	nu_On:			CustomPhase (table:=ADR(phasesTable)):=			(phaseNumber:=24);
	flag1:BOOL;
	Start_AO_From:			CustomPhase (table:=ADR(phasesTable)):=			(phaseNumber:=25);
END_VAR

SUPER^();

//////////////Старт смазки кранов 1 и 2///////////////////////////
IF	algoritms.F3.Smazka_1_2 OR (im.kran1.onStatus = statusDualInput.STATUS_ON) OR (im.kran1.onStatus = statusDualInput.STATUS_TRANSITIONAL)
	OR (im.kran2.onStatus = statusDualInput.STATUS_ON) OR (im.kran2.onStatus = statusDualInput.STATUS_TRANSITIONAL)  THEN
	IF	(algoritms.F3.Smazka_1_2 OR (im.kran1.onStatus = statusDualInput.STATUS_ON) OR (im.kran1.onStatus = statusDualInput.STATUS_TRANSITIONAL)) AND (NOT klapan1.start) AND (NOT kran1Close.top) THEN
		klapan1.run ();
	END_IF
	IF	(algoritms.F3.Smazka_1_2 OR (im.kran2.onStatus = statusDualInput.STATUS_ON) OR (im.kran2.onStatus = statusDualInput.STATUS_TRANSITIONAL)) AND (NOT klapan2.start) AND (NOT kran2Close.top) THEN
		klapan2.run ();
	END_IF
	algoritms.F3.Smazka_1_2:=FALSE;
END_IF

//////////////Переставляем краны///////////////////////////
IF	NOT kran6Open.start THEN
	ystavki.Block_kr6_alg.setValue (1);
	IF	im.kran6._cmdreset.IN = FALSE THEN
		ystavki.Block_kr6_alg.setValue (0);
		kran6Open.run(); //открываем карн 6
	END_IF
END_IF

IF	NOT kran4Close.start THEN
	ystavki.Block_kr4_alg.setValue (1);
	IF	im.kran4._cmdreset.IN = FALSE THEN
		ystavki.Block_kr4_alg.setValue (0);
		kran4Close.run(); //закрываем кран 4
	END_IF
END_IF

IF	NOT kran3bOpen.start THEN
	ystavki.Block_kr3b_alg.setValue (1);
	IF	im.kran3b._cmdreset.IN = FALSE THEN
		ystavki.Block_kr3b_alg.setValue (0);
		kran3bOpen.run (); //Открываем кран 3бис
	END_IF
END_IF
protections.p_mvOff.reset ();
protections.p_OFFAvarSwitch.reset();
protections.p_RegVozbOff.reset ();
protections.p_kran1.reset ();
protections.p_kran2.reset ();
mvOff.run(); //отключаем МВ

IF	NOT kran1Close.start THEN
	ystavki.Block_kr1_alg.setValue (1);
	IF	im.kran1._cmdreset.IN = FALSE THEN
		ystavki.Block_kr1_alg.setValue (0);
		kran1Close.run(); //закрываем кран 1
	END_IF
END_IF

IF	NOT	kran2Close.start THEN
	ystavki.Block_kr2_alg.setValue (1);
	IF	im.kran2._cmdreset.IN = FALSE THEN
		ystavki.Block_kr2_alg.setValue (0);
		kran2Close.run(); //закрываем кран 2 
	END_IF
END_IF

IF	NOT	kran3Close.start THEN
	ystavki.Block_kr3_alg.setValue (1);
	IF	im.kran3._cmdreset.IN = FALSE THEN
		ystavki.Block_kr3_alg.setValue (0);
		kran3Close.run(); //закрываем кран 3
	END_IF
END_IF

IF	kran6Open.top THEN
	algoritms.S_Vibr.CanRun:=FALSE;
	algoritms.S_Vibr.reset ();
END_IF
///////////////выдаем смазку кранов 1 и 2//////////////////////////
IF	klapan1.start AND kran1Close.top THEN
	im.Kr1_Smazka.impulse();//выдача команды на клапан
	klapan1.top:=TRUE;
END_IF;
IF	klapan2.start AND kran2Close.top THEN
	im.Kr2_Smazka.impulse();//выдача команды на клапан
	klapan2.top:=TRUE;
END_IF;
///////////////открываем кран 5//////////////////////////
IF 	kran1Close.top AND kran2Close.top AND kran3Close.top AND kran4Close.top AND NOT kran5Open.top THEN //если кран 1 и 2 закрыты открываем кран 5
	IF	NOT	kran5Open.start THEN
		ystavki.Block_kr5_alg.setValue (1);
		IF	im.kran5._cmdreset.IN = FALSE THEN
			ystavki.Block_kr5_alg.setValue (0);
			kran5Open.run();
		END_IF
	END_IF

	//protections.p_DGazaNaVhodeNagnetatelja.reset ();
	protections.p_DGazaNaVyhodeNagnetatelja.reset ();
END_IF 
/////////////////////////////////////////
IF	mvOff.top AND NOT flag1 THEN //если МВ отключился 
	algoritms.AutoPNS_Start.canrun :=FALSE;
	algoritms.AutoPNS_Start.reset ();
	algoritms.autoPns.canrun :=FALSE;
	autoPnsOff.run ();
	pnsOn.run ();
	nu_On.run();
	CASE 	im.nu.mainNasos.Value OF
	0:		im.nu.nu1.on ();
	1:		im.nu.nu2.on ();
	END_CASE
	algoritms.autoNu_2.canrun:=FALSE;
	algoritms.autoNu_2.reset ();
	algoritms.autoNu_1.canrun:=TRUE;
	algoritms.autoNu_1.run ();
	flag1:=TRUE;
END_IF
IF	((im.nu.nu1.onStatus =statusDualInput.STATUS_On) OR (im.nu.nu2.onStatus =statusDualInput.STATUS_On)) AND nu_On.start AND NOT nu_On.top THEN
	nu_On.top:=TRUE;
END_IF
/////////////////////////////////////////
IF 	kran5Open.top THEN //если отключены МВ и 5 кран
	Pg_VhodLessThen300.run();  //проверяем условие, что давление в нагнетателе меньше 100
	Pg_VyhodLessThen300.run(); 
	
END_IF 
/////////////////////////////////////////
IF Pg_VhodLessThen300.start AND (NOT Pg_VhodLessThen300.top) THEN
	IF 	(ai.DGazaNaVhodeNagnetatelja.interval>=statusAi.NORMAL) AND (ai.DGazaNaVhodeNagnetatelja.value < 0.3 )THEN
		Pg_VhodLessThen300.top:=TRUE; //давление в полости нагнетателя меньше 100 кПа
	END_IF
END_IF
/////////////////////////////////////////
IF Pg_VyhodLessThen300.start AND (NOT Pg_VyhodLessThen300.top) THEN
	IF 	(ai.DGazaNaVyhodeNagnetatelja.interval>=statusAi.NORMAL) AND (ai.DGazaNaVyhodeNagnetatelja.value < 0.3) THEN
		Pg_VyhodLessThen300.top:=TRUE; //давление в полости нагнетателя меньше 100 кПа
	END_IF
END_IF
/////////////////////////////////////////
IF 	Pg_VhodLessThen300.top AND Pg_VyhodLessThen300.top AND pnsOn.top AND nu_On.top AND mvOff.top THEN //давление меньше 100 и кран5 и пнс включен 
	nuOff.run(); //отключаем НУ
	protections.p_PerepadDavlenieMasloGaz.reset();
	protections.p_PerepadDavlenieMasloGaz_Less100.reset();
	
	protections.p_DGazaNaVhodeNagnetatelja_GPA_STOP.run ();
	protections.p_DGazaNaVyhodeNagnetatelja_GPA_STOP.run ();
	Auto_NU_Off.top:=TRUE;
	algoritms.autoNu_1.CanRun:=FALSE;
	algoritms.autoNu_1.reset ();
END_IF
/////////////////////////////////////////
IF	nuOff.top THEN //при отключенном ну можо сбросить выбег
	IF	NOT algmanager.reg_V AND NOT pnsoff.start THEN
		timer600.run();
	END_IF;
	IF	NOT pnsoff.start THEN
		sbrosVibeg.ask();
	END_IF;
END_IF
/////////////////////////////////////////
IF 	((timer600.top) OR (sbrosVibeg.answer=Answers.ANS_YES))   THEN //Если прошло 480 секунд и НУ выключен или нажата сброс выбега
	pnsOff.run();//отключаем ПНС
	protections.p_DavlenijaMasloSmNizkoe.reset ();
	protections.p_DavlenijaMasloSmVysokoe.reset ();
	sbrosVibeg.reset ();
	timer600.reset ();
	algoritms.F2_Ch.autoAVOM_canrun_flag:=FALSE;
	algoritms.F2_R.autoAVOM_canrun_flag:=FALSE;
END_IF
IF	(NOT algoritms.F2_Ch.autoAVOM_canrun_flag) AND (NOT algoritms.F2_R.autoAVOM_canrun_flag) AND pnsoff.start THEN
	Avom1Off.run ();
	Avom2Off.run ();
	Avom3Off.run ();
	Avom4Off.run ();
	algoritms.R_AutoAVOM.CanRun:=FALSE;
	algoritms.R_AutoAVOM.reset();
	algoritms.S_AutoAVOM.CanRun:=FALSE;
	algoritms.S_AutoAVOM.reset();
	algoritms.Auto_Avom_.CanRun:=FALSE;
	autoAVOMOff.run ();
END_IF
/////////////////////////////////////////
IF 	pnsOff.top AND Avom1Off.top AND Avom2Off.top AND Avom3Off.top AND Avom4Off.top AND autoAVOMOff.top  THEN //Если  отключен ПНС завершаем алгоритм
	end();
	timer5.run ();
END_IF
/////////////////////////////////////////
IF 	timer5.top THEN
	timer5.reset ();
	reset ();
END_IF

METHOD PUBLIC reset
VAR_INPUT
END_VAR
SUPER^.reset();
sbrosVibeg.reset();
statusSet.setBit(15,0);
flag1:=FALSE;
ystavki.Block_kr1_alg.setValue (0);
ystavki.Block_kr2_alg.setValue (0);
END_METHOD

METHOD PUBLIC run
VAR_INPUT
END_VAR
SUPER^.run();
algManager.setMode(nMode:=ModeGpa.MODE_AO);
statusSet.setBit(15,1);
IF	algmanager.reg_V THEN
	Start_AO_From.top:=TRUE;
END_IF
END_METHOD

END_FUNCTION_BLOCK

// lowLevel_ecl/algoritms/phases/ph_Kran
	{attribute 'symbol' := 'none'}
FUNCTION_BLOCK ph_Kran EXTENDS BaseAlgoritmPhase
VAR_INPUT
	im:REFERENCE TO DualStateKran;
	act:DualStateImAction;
END_VAR
VAR_OUTPUT
END_VAR
VAR
END_VAR

SUPER^();

METHOD PROTECTED getError : bool
VAR_INPUT
END_VAR
getError:=Im.CommandFail();
END_METHOD

METHOD protected GetIm : POINTER TO BaseIm
VAR_INPUT
END_VAR
GetIm:=adr(Im);
END_METHOD

METHOD PROTECTED getTop : bool
VAR_INPUT
END_VAR
CASE act OF
	DualStateImAction.on:
		getTop:=Im.onStatus=statusDualInput.STATUS_ON;
	DualStateImAction.off:
		getTop:=Im.onStatus=statusDualInput.STATUS_OFF;
END_CASE;
END_METHOD

METHOD PROTECTED onRun
VAR_INPUT
END_VAR

CASE act OF
	DualStateImAction.on:
		Im.open();
	DualStateImAction.off:
		Im.close();
END_CASE
END_METHOD

END_FUNCTION_BLOCK

// lowLevel_ecl/algoritms/phases/ph_Switch
	{attribute 'symbol' := 'none'}
FUNCTION_BLOCK ph_Switch EXTENDS BaseAlgoritmPhase
VAR_INPUT
	Im:REFERENCE TO DualStateSwitch;
	act:DualStateImAction;
END_VAR
VAR_OUTPUT
END_VAR
VAR
END_VAR

SUPER^();

METHOD PROTECTED getError : bool
VAR_INPUT
END_VAR
getError:=Im.CommandFail();
END_METHOD

METHOD protected GetIm : POINTER TO BaseIm
VAR_INPUT
END_VAR
GetIm:=adr(Im);
END_METHOD

METHOD PROTECTED getTop : bool
VAR_INPUT
END_VAR
CASE act OF
	DualStateImAction.on:
		getTop:=Im.onStatus=statusDualInput.STATUS_ON;
	DualStateImAction.off:
		getTop:=Im.onStatus=statusDualInput.STATUS_OFF;
END_CASE;
END_METHOD

METHOD PROTECTED onRun
VAR_INPUT
END_VAR
CASE act OF
	DualStateImAction.on:
		Im.on();
	DualStateImAction.off:
		Im.off();
END_CASE
END_METHOD

END_FUNCTION_BLOCK

// lowLevel_ecl/algoritms/phases/ph_algoritm
	{attribute 'symbol' := 'none'}
FUNCTION_BLOCK ph_algoritm EXTENDS BaseAlgoritmPhase
VAR_INPUT
	Im:REFERENCE TO BaseAlgoritm;
	act:PhaseAlgoritmAction; // run reset
	waitCompletion:BOOL;
END_VAR
VAR_OUTPUT
END_VAR
VAR
END_VAR

SUPER^();

METHOD PROTECTED getError : bool
VAR_INPUT
END_VAR
getError:=Im.hasError OR Im.CommandFail();
END_METHOD

METHOD protected GetIm : POINTER TO BaseIm
VAR_INPUT
END_VAR
GetIm:=ADR(Im);
END_METHOD

METHOD PROTECTED getTop : bool
VAR_INPUT
END_VAR
CASE act OF
	PhaseAlgoritmAction.run:
		IF waitCompletion THEN
			getTop:=Im.isEnded;
		ELSE
			getTop:=Im.isRuning;			
		END_IF
	PhaseAlgoritmAction.reset:
		getTop:=NOT Im.isRuning;
END_CASE
END_METHOD

METHOD PROTECTED onRun
VAR_INPUT
END_VAR
CASE act OF
	PhaseAlgoritmAction.run:
		Im.run();
	PhaseAlgoritmAction.reset:
		Im.reset();
END_CASE
END_METHOD

END_FUNCTION_BLOCK

// K1/std12k5/ostanov/noAlg
	{attribute 'symbol' := 'none'}
FUNCTION_BLOCK noAlg EXTENDS StepBySteapAlgoritm
VAR_INPUT
END_VAR
VAR_OUTPUT
{attribute 'symbol' := 'read'}
	sbrosVibeg:		Question(table:=ADR(ObjectTable)):=			(AnswerVariants:=Answers.ANS_YES);
END_VAR
VAR
	{attribute 'symbol' := 'read'}
	timer120:		ph_Timer (table:=ADR(phasesTable)):=			(phaseNumber:=0, delay:=T#120S);
	
	kran6Open:		ph_Kran (table:=ADR(phasesTable)):=				(phaseNumber:=1, Im:=Im.kran6, act:=DualStateImAction.on);
	
	kran4Close:		ph_Kran (table:=ADR(phasesTable)):=				(phaseNumber:=2, Im:=Im.kran4, act:=DualStateImAction.off);
	
	kran3bOpen:		ph_Kran (table:=ADR(phasesTable)):=				(phaseNumber:=3, Im:=Im.kran3b, act:=DualStateImAction.on);
	
	mvOff:			ph_Switch (table:=ADR(phasesTable)):=			(phaseNumber:=4, Im:=Im.mv, act:=DualStateImAction.off);
	
	kran1Close:		ph_Kran (table:=ADR(phasesTable)):=				(phaseNumber:=5, Im:=Im.kran1, act:=DualStateImAction.off);
	
	kran2Close:		ph_Kran (table:=ADR(phasesTable)):=				(phaseNumber:=6, Im:=Im.kran2, act:=DualStateImAction.off);
	
	kran3Close:		ph_Kran (table:=ADR(phasesTable)):=				(phaseNumber:=7, Im:=Im.kran3, act:=DualStateImAction.off);
	
	kran5Open:		ph_Kran (table:=ADR(phasesTable)):=				(phaseNumber:=8, Im:=Im.kran5, act:=DualStateImAction.on);
	
	error_Krans:	CustomPhase (table:=ADR(phasesTable)):=			(phaseNumber:=9);
	
	autoPnsOff:		ph_algoritm (table:=ADR(phasesTable)):=			(phaseNumber:=10, Im:=algoritms.autoPns, act:=PhaseAlgoritmAction.reset, waitCompletion:=FALSE);
	
	pnsOn:			ph_Switch (table:=ADR(phasesTable)):=			(phaseNumber:=11, Im:=Im.pns, act:=DualStateImAction.on);
	
	Pg_VhodLessThen300:	CustomPhase (table:=ADR(phasesTable)):=		(phaseNumber:=12);
	
	Pg_VyhodLessThen300:CustomPhase (table:=ADR(phasesTable)):=		(phaseNumber:=13);
	
	nuOff:			ph_Switch  (table:=ADR(phasesTable)):=			(phaseNumber:=14, Im:=Im.nu, act:=DualStateImAction.off);
	AutoNU_Off:		CustomPhase (table:=ADR(phasesTable)):=		(phaseNumber:=15);
	{attribute 'symbol' := 'read'}
	timer600:		ph_Timer (table:=ADR(phasesTable)):=			(phaseNumber:=16, delay:=T#600S);
	
	pnsOff:			ph_Switch (table:=ADR(phasesTable)):=			(phaseNumber:=17, Im:=Im.pns, act:=DualStateImAction.off);
	
	Avom1Off:		ph_Switch (table:=ADR(phasesTable)):=			(phaseNumber:=18, Im:=Im.v1_Avom, act:=DualStateImAction.off);
	
	Avom2Off:		ph_Switch (table:=ADR(phasesTable)):=			(phaseNumber:=19, Im:=Im.v2_Avom, act:=DualStateImAction.off);
	
	Avom3Off:		ph_Switch (table:=ADR(phasesTable)):=			(phaseNumber:=20, Im:=Im.v3_Avom, act:=DualStateImAction.off);
	
	Avom4Off:		ph_Switch (table:=ADR(phasesTable)):=			(phaseNumber:=21, Im:=Im.v4_Avom, act:=DualStateImAction.off);
	
	autoAVOMOff:	ph_algoritm (table:=ADR(phasesTable)):=			(phaseNumber:=22, Im:=algoritms.Auto_Avom_, act:=PhaseAlgoritmAction.reset, waitCompletion:=FALSE);
	
	timer5:			ph_Timer (table:=ADR(phasesTable)):=			(phaseNumber:=23, delay:=T#5S);
	
	klapan1:		CustomPhase (table:=ADR(phasesTable)):=			(phaseNumber:=24);
	
	klapan2:		CustomPhase (table:=ADR(phasesTable)):=			(phaseNumber:=25);
	
	nu_On:			CustomPhase (table:=ADR(phasesTable)):=			(phaseNumber:=26);
	flag1:bool;
END_VAR

SUPER^();
///////////////Счетчик//////////////////////////
IF	NOT kran6Open.top AND NOT timer120.top  THEN //Если кран 5 не открыт
	timer120.run (); //запускаем счетчик 480 сек
ELSE
	IF	timer120.top AND NOT kran6Open.top THEN //если счетчик отсчитал и кран 5 не открыт, то выставляем ошибку фазы
		error_Krans.error := TRUE;
	END_IF;
END_IF
//////////////Старт смазки кранов 1 и 2///////////////////////////
IF	algoritms.F3.Smazka_1_2 OR (im.kran1.onStatus = statusDualInput.STATUS_ON) OR (im.kran1.onStatus = statusDualInput.STATUS_TRANSITIONAL)
	OR (im.kran2.onStatus = statusDualInput.STATUS_ON) OR (im.kran2.onStatus = statusDualInput.STATUS_TRANSITIONAL)  THEN
	IF	(algoritms.F3.Smazka_1_2 OR (im.kran1.onStatus = statusDualInput.STATUS_ON) OR (im.kran1.onStatus = statusDualInput.STATUS_TRANSITIONAL)) AND (NOT klapan1.start) AND (NOT kran1Close.top) THEN
		klapan1.run ();
	END_IF
	IF	(algoritms.F3.Smazka_1_2 OR (im.kran2.onStatus = statusDualInput.STATUS_ON) OR (im.kran2.onStatus = statusDualInput.STATUS_TRANSITIONAL)) AND (NOT klapan2.start) AND (NOT kran2Close.top) THEN
		klapan2.run ();
	END_IF
	algoritms.F3.Smazka_1_2:=FALSE;
END_IF
//////////////Переставляем краны///////////////////////////
kran6Open.run(); //открываем карн 6
kran4Close.run(); //закрываем кран 4
IF kran4Close.top THEN
ystavki.Block_kr4_alg.setValue (0);
END_IF
IF	kran6Open.top THEN
	kran3bOpen.run (); //Открываем кран 3бис
	timer120.reset (); 
	error_Krans.top := FALSE;
	error_Krans.error := FALSE;
	algoritms.S_Vibr.CanRun:=FALSE;
	algoritms.S_Vibr.reset ();
END_IF
IF	kran3bOpen.top AND NOT mvoff.start THEN
	protections.p_mvOff.reset ();
	protections.p_OFFAvarSwitch.reset();
	protections.p_RegVozbOff.reset ();
	mvOff.run(); //отключаем МВ
END_IF;
/////////////////////////////////////////
IF	mvOff.top AND NOT flag1 THEN //если МВ отключился 
	algoritms.AutoPNS_Start.canrun :=FALSE;
	algoritms.AutoPNS_Start.reset ();
	algoritms.autoPns.canrun :=FALSE;
	autoPnsOff.run ();
	pnsOn.run ();
	protections.p_kran1.reset ();
	protections.p_kran2.reset ();
	kran1Close.run(); //закрываем кран 1
	kran2Close.run(); //закрываем кран 2
	kran3Close.run(); //закрываем кран 3
	nu_On.run();
	CASE 	im.nu.mainNasos.Value OF
	0:		im.nu.nu1.on ();
	1:		im.nu.nu2.on ();
	END_CASE
	algoritms.autoNu_2.canrun:=FALSE;
	algoritms.autoNu_2.reset ();
	algoritms.autoNu_1.canrun:=TRUE;
	algoritms.autoNu_1.run ();
	flag1:=TRUE;
END_IF
IF	((im.nu.nu1.onStatus =statusDualInput.STATUS_On) OR (im.nu.nu2.onStatus =statusDualInput.STATUS_On)) AND nu_On.start AND NOT nu_On.top THEN
	nu_On.top:=TRUE;
END_IF

///////////////выдаем смазку кранов 1 и 2//////////////////////////
IF	klapan1.start AND kran1Close.top THEN
	im.Kr1_Smazka.impulse();//выдача команды на клапан
	klapan1.top:=TRUE;
END_IF;
IF	klapan2.start AND kran2Close.top THEN
	im.Kr2_Smazka.impulse();//выдача команды на клапан
	klapan2.top:=TRUE;
END_IF;
///////////////открываем кран 5//////////////////////////
IF 	kran1Close.top AND kran2Close.top AND kran3Close.top AND kran4Close.top THEN //если кран 1 и 2 закрыты открываем кран 5
	kran5Open.run();
	//protections.p_DGazaNaVhodeNagnetatelja.reset ();
	protections.p_DGazaNaVyhodeNagnetatelja.reset ();
END_IF 


/////////////////////////////////////////
IF 	kran5Open.top THEN //если отключены МВ и 5 кран
	Pg_VhodLessThen300.run();  //проверяем условие, что давление в нагнетателе меньше 100
	Pg_VyhodLessThen300.run(); 
	
END_IF 
/////////////////////////////////////////
IF Pg_VhodLessThen300.start AND (NOT Pg_VhodLessThen300.top) THEN
	IF 	(ai.DGazaNaVhodeNagnetatelja.interval>=statusAi.NORMAL) AND (ai.DGazaNaVhodeNagnetatelja.value < 0.3) THEN
		Pg_VhodLessThen300.top:=TRUE; //давление в полости нагнетателя меньше 100 кПа
	END_IF
END_IF
/////////////////////////////////////////
IF Pg_VyhodLessThen300.start AND (NOT Pg_VyhodLessThen300.top) THEN
	IF 	(ai.DGazaNaVyhodeNagnetatelja.interval>=statusAi.NORMAL )AND (ai.DGazaNaVyhodeNagnetatelja.value < 0.3) THEN
		Pg_VyhodLessThen300.top:=TRUE; //давление в полости нагнетателя меньше 100 кПа
	END_IF
END_IF
/////////////////////////////////////////
IF 	Pg_VhodLessThen300.top AND Pg_VyhodLessThen300.top AND pnsOn.top AND nu_On.top AND mvOff.top  THEN //давление меньше 100 и кран5 и пнс включен 
	nuOff.run(); //отключаем НУ
	protections.p_PerepadDavlenieMasloGaz.reset();
	protections.p_PerepadDavlenieMasloGaz_Less100.reset();
	
	protections.p_DGazaNaVhodeNagnetatelja_GPA_STOP.run ();
	protections.p_DGazaNaVyhodeNagnetatelja_GPA_STOP.run ();
	algoritms.autoNu_1.CanRun:=FALSE;
	AutoNU_Off.top:=TRUE;
	algoritms.autoNu_1.reset ();
END_IF
/////////////////////////////////////////
IF	nuOff.top THEN //при отключенном ну можо сбросить выбег
	IF	NOT algmanager.reg_V AND NOT pnsoff.start THEN
		timer600.run();
	END_IF;
	IF	NOT pnsoff.start THEN
		sbrosVibeg.ask();
	END_IF;
END_IF
/////////////////////////////////////////
IF 	((timer600.top) OR (sbrosVibeg.answer=Answers.ANS_YES))   THEN //Если прошло 480 секунд и НУ выключен или нажата сброс выбега
	pnsOff.run();//отключаем ПНС
	protections.p_DavlenijaMasloSmNizkoe.reset ();
	protections.p_DavlenijaMasloSmVysokoe.reset ();
	sbrosVibeg.reset ();
	timer600.reset ();
	algoritms.F2_Ch.autoAVOM_canrun_flag:=FALSE;
	algoritms.F2_R.autoAVOM_canrun_flag:=FALSE;
END_IF
IF	(NOT algoritms.F2_Ch.autoAVOM_canrun_flag) AND (NOT algoritms.F2_R.autoAVOM_canrun_flag) AND pnsoff.start THEN
	Avom1Off.run ();
	Avom2Off.run ();
	Avom3Off.run ();
	Avom4Off.run ();
	algoritms.R_AutoAVOM.CanRun:=FALSE; 
	algoritms.R_AutoAVOM.reset();
	algoritms.S_AutoAVOM.CanRun:=FALSE;
	algoritms.S_AutoAVOM.reset();
	algoritms.Auto_Avom_.CanRun:=FALSE;
	autoAVOMOff.run ();
END_IF
/////////////////////////////////////////
IF 	pnsOff.top AND Avom1Off.top AND Avom2Off.top AND Avom3Off.top AND Avom4Off.top AND autoAVOMOff.top  THEN //Если  отключен ПНС завершаем алгоритм
	end();
	timer5.run ();
END_IF
/////////////////////////////////////////
IF 	timer5.top THEN
	timer5.reset ();
	reset ();
END_IF

METHOD PUBLIC reset
VAR_INPUT
END_VAR
SUPER^.reset();
sbrosVibeg.reset();
statusSet.setBit(15,0);
flag1:=FALSE;
END_METHOD

METHOD PUBLIC run
VAR_INPUT
END_VAR
SUPER^.run();
algManager.setMode(nMode:=ModeGpa.MODE_NO);
statusSet.setBit(15,1);
END_METHOD

END_FUNCTION_BLOCK

// K2/std12k5/ostanov/noAlg
	{attribute 'symbol' := 'none'}
FUNCTION_BLOCK noAlg EXTENDS StepBySteapAlgoritm
VAR_INPUT
END_VAR
VAR_OUTPUT
{attribute 'symbol' := 'read'}
	sbrosVibeg:		Question(table:=ADR(ObjectTable)):=			(AnswerVariants:=Answers.ANS_YES);
END_VAR
VAR
	{attribute 'symbol' := 'read'}
	timer120:		ph_Timer (table:=ADR(phasesTable)):=			(phaseNumber:=0, delay:=T#120S);
	
	kran6Open:		ph_Kran (table:=ADR(phasesTable)):=				(phaseNumber:=1, Im:=Im.kran6, act:=DualStateImAction.on);
	
	kran4Close:		ph_Kran (table:=ADR(phasesTable)):=				(phaseNumber:=2, Im:=Im.kran4, act:=DualStateImAction.off);
	
	kran3bOpen:		ph_Kran (table:=ADR(phasesTable)):=				(phaseNumber:=3, Im:=Im.kran3b, act:=DualStateImAction.on);
	
	mvOff:			ph_Switch (table:=ADR(phasesTable)):=			(phaseNumber:=4, Im:=Im.mv, act:=DualStateImAction.off);
	
	kran1Close:		ph_Kran (table:=ADR(phasesTable)):=				(phaseNumber:=5, Im:=Im.kran1, act:=DualStateImAction.off);
	
	kran2Close:		ph_Kran (table:=ADR(phasesTable)):=				(phaseNumber:=6, Im:=Im.kran2, act:=DualStateImAction.off);
	
	kran3Close:		ph_Kran (table:=ADR(phasesTable)):=				(phaseNumber:=7, Im:=Im.kran3, act:=DualStateImAction.off);
	
	kran5Open:		ph_Kran (table:=ADR(phasesTable)):=				(phaseNumber:=8, Im:=Im.kran5, act:=DualStateImAction.on);
	
	error_Krans:	CustomPhase (table:=ADR(phasesTable)):=			(phaseNumber:=9);
	
	autoPnsOff:		ph_algoritm (table:=ADR(phasesTable)):=			(phaseNumber:=10, Im:=algoritms.autoPns, act:=PhaseAlgoritmAction.reset, waitCompletion:=FALSE);
	
	pnsOn:			ph_Switch (table:=ADR(phasesTable)):=			(phaseNumber:=11, Im:=Im.pns, act:=DualStateImAction.on);
	
	Pg_VhodLessThen300:	CustomPhase (table:=ADR(phasesTable)):=		(phaseNumber:=12);
	
	Pg_VyhodLessThen300:CustomPhase (table:=ADR(phasesTable)):=		(phaseNumber:=13);
	
	nuOff:			ph_Switch  (table:=ADR(phasesTable)):=			(phaseNumber:=14, Im:=Im.nu, act:=DualStateImAction.off);
	AutoNU_Off:		CustomPhase (table:=ADR(phasesTable)):=		(phaseNumber:=15);
	{attribute 'symbol' := 'read'}
	timer600:		ph_Timer (table:=ADR(phasesTable)):=			(phaseNumber:=16, delay:=T#600S);
	
	pnsOff:			ph_Switch (table:=ADR(phasesTable)):=			(phaseNumber:=17, Im:=Im.pns, act:=DualStateImAction.off);
	
	Avom1Off:		ph_Switch (table:=ADR(phasesTable)):=			(phaseNumber:=18, Im:=Im.v1_Avom, act:=DualStateImAction.off);
	
	Avom2Off:		ph_Switch (table:=ADR(phasesTable)):=			(phaseNumber:=19, Im:=Im.v2_Avom, act:=DualStateImAction.off);
	
	Avom3Off:		ph_Switch (table:=ADR(phasesTable)):=			(phaseNumber:=20, Im:=Im.v3_Avom, act:=DualStateImAction.off);
	
	Avom4Off:		ph_Switch (table:=ADR(phasesTable)):=			(phaseNumber:=21, Im:=Im.v4_Avom, act:=DualStateImAction.off);
	
	autoAVOMOff:	ph_algoritm (table:=ADR(phasesTable)):=			(phaseNumber:=22, Im:=algoritms.Auto_Avom_, act:=PhaseAlgoritmAction.reset, waitCompletion:=FALSE);
	
	timer5:			ph_Timer (table:=ADR(phasesTable)):=			(phaseNumber:=23, delay:=T#5S);
	
	klapan1:		CustomPhase (table:=ADR(phasesTable)):=			(phaseNumber:=24);
	
	klapan2:		CustomPhase (table:=ADR(phasesTable)):=			(phaseNumber:=25);
	
	nu_On:			CustomPhase (table:=ADR(phasesTable)):=			(phaseNumber:=26);
	flag1:bool;
END_VAR

SUPER^();
///////////////Счетчик//////////////////////////
IF	NOT kran6Open.top AND NOT timer120.top  THEN //Если кран 5 не открыт
	timer120.run (); //запускаем счетчик 480 сек
ELSE
	IF	timer120.top AND NOT kran6Open.top THEN //если счетчик отсчитал и кран 5 не открыт, то выставляем ошибку фазы
		error_Krans.error := TRUE;
	END_IF;
END_IF
//////////////Старт смазки кранов 1 и 2///////////////////////////
IF	algoritms.F3.Smazka_1_2 OR (im.kran1.onStatus = statusDualInput.STATUS_ON) OR (im.kran1.onStatus = statusDualInput.STATUS_TRANSITIONAL)
	OR (im.kran2.onStatus = statusDualInput.STATUS_ON) OR (im.kran2.onStatus = statusDualInput.STATUS_TRANSITIONAL)  THEN
	IF	(algoritms.F3.Smazka_1_2 OR (im.kran1.onStatus = statusDualInput.STATUS_ON) OR (im.kran1.onStatus = statusDualInput.STATUS_TRANSITIONAL)) AND (NOT klapan1.start) AND (NOT kran1Close.top) THEN
		klapan1.run ();
	END_IF
	IF	(algoritms.F3.Smazka_1_2 OR (im.kran2.onStatus = statusDualInput.STATUS_ON) OR (im.kran2.onStatus = statusDualInput.STATUS_TRANSITIONAL)) AND (NOT klapan2.start) AND (NOT kran2Close.top) THEN
		klapan2.run ();
	END_IF
	algoritms.F3.Smazka_1_2:=FALSE;
END_IF
//////////////Переставляем краны///////////////////////////
kran6Open.run(); //открываем карн 6
kran4Close.run(); //закрываем кран 4
IF kran4Close.top THEN
ystavki.Block_kr4_alg.setValue (0);
END_IF
IF	kran6Open.top THEN
	kran3bOpen.run (); //Открываем кран 3бис
	timer120.reset (); 
	error_Krans.top := FALSE;
	error_Krans.error := FALSE;
	algoritms.S_Vibr.CanRun:=FALSE;
	algoritms.S_Vibr.reset ();
END_IF
IF	kran3bOpen.top AND NOT mvoff.start THEN
	protections.p_mvOff.reset ();
	protections.p_OFFAvarSwitch.reset();
	protections.p_RegVozbOff.reset ();
	mvOff.run(); //отключаем МВ
END_IF;
/////////////////////////////////////////
IF	mvOff.top AND NOT flag1 THEN //если МВ отключился 
	algoritms.AutoPNS_Start.canrun :=FALSE;
	algoritms.AutoPNS_Start.reset ();
	algoritms.autoPns.canrun :=FALSE;
	autoPnsOff.run ();
	pnsOn.run ();
	protections.p_kran1.reset ();
	protections.p_kran2.reset ();
	kran1Close.run(); //закрываем кран 1
	kran2Close.run(); //закрываем кран 2
	kran3Close.run(); //закрываем кран 3
	nu_On.run();
	CASE 	im.nu.mainNasos.Value OF
	0:		im.nu.nu1.on ();
	1:		im.nu.nu2.on ();
	END_CASE
	algoritms.autoNu_2.canrun:=FALSE;
	algoritms.autoNu_2.reset ();
	algoritms.autoNu_1.canrun:=TRUE;
	algoritms.autoNu_1.run ();
	flag1:=TRUE;
END_IF
IF	((im.nu.nu1.onStatus =statusDualInput.STATUS_On) OR (im.nu.nu2.onStatus =statusDualInput.STATUS_On)) AND nu_On.start AND NOT nu_On.top THEN
	nu_On.top:=TRUE;
END_IF

///////////////выдаем смазку кранов 1 и 2//////////////////////////
IF	klapan1.start AND kran1Close.top THEN
	im.Kr1_Smazka.impulse();//выдача команды на клапан
	klapan1.top:=TRUE;
END_IF;
IF	klapan2.start AND kran2Close.top THEN
	im.Kr2_Smazka.impulse();//выдача команды на клапан
	klapan2.top:=TRUE;
END_IF;
///////////////открываем кран 5//////////////////////////
IF 	kran1Close.top AND kran2Close.top AND kran3Close.top AND kran4Close.top THEN //если кран 1 и 2 закрыты открываем кран 5
	kran5Open.run();
	//protections.p_DGazaNaVhodeNagnetatelja.reset ();
	protections.p_DGazaNaVyhodeNagnetatelja.reset ();
END_IF 


/////////////////////////////////////////
IF 	kran5Open.top THEN //если отключены МВ и 5 кран
	Pg_VhodLessThen300.run();  //проверяем условие, что давление в нагнетателе меньше 100
	Pg_VyhodLessThen300.run(); 
	
END_IF 
/////////////////////////////////////////
IF Pg_VhodLessThen300.start AND (NOT Pg_VhodLessThen300.top) THEN
	IF 	(ai.DGazaNaVhodeNagnetatelja.interval>=statusAi.NORMAL) AND (ai.DGazaNaVhodeNagnetatelja.value < 0.3) THEN
		Pg_VhodLessThen300.top:=TRUE; //давление в полости нагнетателя меньше 100 кПа
	END_IF
END_IF
/////////////////////////////////////////
IF Pg_VyhodLessThen300.start AND (NOT Pg_VyhodLessThen300.top) THEN
	IF 	(ai.DGazaNaVyhodeNagnetatelja.interval>=statusAi.NORMAL )AND (ai.DGazaNaVyhodeNagnetatelja.value < 0.3) THEN
		Pg_VyhodLessThen300.top:=TRUE; //давление в полости нагнетателя меньше 100 кПа
	END_IF
END_IF
/////////////////////////////////////////
IF 	Pg_VhodLessThen300.top AND Pg_VyhodLessThen300.top AND pnsOn.top AND nu_On.top AND mvOff.top  THEN //давление меньше 100 и кран5 и пнс включен 
	nuOff.run(); //отключаем НУ
	protections.p_PerepadDavlenieMasloGaz.reset();
	protections.p_PerepadDavlenieMasloGaz_Less100.reset();
	
	protections.p_DGazaNaVhodeNagnetatelja_GPA_STOP.run ();
	protections.p_DGazaNaVyhodeNagnetatelja_GPA_STOP.run ();
	algoritms.autoNu_1.CanRun:=FALSE;
	AutoNU_Off.top:=TRUE;
	algoritms.autoNu_1.reset ();
END_IF
/////////////////////////////////////////
IF	nuOff.top THEN //при отключенном ну можо сбросить выбег
	IF	NOT algmanager.reg_V AND NOT pnsoff.start THEN
		timer600.run();
	END_IF;
	IF	NOT pnsoff.start THEN
		sbrosVibeg.ask();
	END_IF;
END_IF
/////////////////////////////////////////
IF 	((timer600.top) OR (sbrosVibeg.answer=Answers.ANS_YES))   THEN //Если прошло 480 секунд и НУ выключен или нажата сброс выбега
	pnsOff.run();//отключаем ПНС
	protections.p_DavlenijaMasloSmNizkoe.reset ();
	protections.p_DavlenijaMasloSmVysokoe.reset ();
	sbrosVibeg.reset ();
	timer600.reset ();
	algoritms.F2_Ch.autoAVOM_canrun_flag:=FALSE;
	algoritms.F2_R.autoAVOM_canrun_flag:=FALSE;
END_IF
IF	(NOT algoritms.F2_Ch.autoAVOM_canrun_flag) AND (NOT algoritms.F2_R.autoAVOM_canrun_flag) AND pnsOff.start THEN
	Avom1Off.run ();
	Avom2Off.run ();
	Avom3Off.run ();
	Avom4Off.run ();
	algoritms.R_AutoAVOM.CanRun:=FALSE; 
	algoritms.R_AutoAVOM.reset();
	algoritms.S_AutoAVOM.CanRun:=FALSE;
	algoritms.S_AutoAVOM.reset();
	algoritms.Auto_Avom_.CanRun:=FALSE;
	autoAVOMOff.run ();
END_IF
/////////////////////////////////////////
IF 	pnsOff.top AND Avom1Off.top AND Avom2Off.top AND Avom3Off.top AND Avom4Off.top AND autoAVOMOff.top  THEN //Если  отключен ПНС завершаем алгоритм
	end();
	timer5.run ();
END_IF
/////////////////////////////////////////
IF 	timer5.top THEN
	timer5.reset ();
	reset ();
END_IF

METHOD PUBLIC reset
VAR_INPUT
END_VAR
SUPER^.reset();
sbrosVibeg.reset();
statusSet.setBit(15,0);
flag1:=FALSE;
END_METHOD

METHOD PUBLIC run
VAR_INPUT
END_VAR
SUPER^.run();
algManager.setMode(nMode:=ModeGpa.MODE_NO);
statusSet.setBit(15,1);
END_METHOD

END_FUNCTION_BLOCK

// K1/std12k5/Prov/Opressovka
{attribute 'symbol' := 'none'}
FUNCTION_BLOCK Opressovka EXTENDS StepBySteapAlgoritm
VAR_INPUT
	{attribute 'symbol' := 'read'}
	Auto:DiscretParametr(table:=ADR(objectTable));//{name:Автоматический или ручной режим работы}
	{attribute 'symbol' := 'read'}
	MaxZapolnenie:AnalogParametr(table:=ADR(objectTable));//{name:задайте сюда значение}
END_VAR
VAR_OUTPUT
	{attribute 'symbol' := 'read'}
	Opressovka_Start:		Question(table:=ADR(ObjectTable)):=			(AnswerVariants:=(Answers.ANS_YES OR Answers.ANS_NO));
	{attribute 'symbol' := 'read'}
	PNS_NU_ON_Ask:		Question(table:=ADR(ObjectTable)):=			(AnswerVariants:=Answers.ANS_YES);
	{attribute 'symbol' := 'read'}
	Zapolnit_kontur:	Question(table:=ADR(ObjectTable)):=			(AnswerVariants:=Answers.ANS_YES);
END_VAR
VAR
	OPC_Control:	CustomPhase (table:=ADR(phasesTable)):=		(phaseNumber:=0);
	Pms_more_50:	CustomPhase (table:=ADR(phasesTable)):=		(phaseNumber:=1);
	Pms_more_300:	CustomPhase (table:=ADR(phasesTable)):=		(phaseNumber:=2);
	dPmg_more_100:	CustomPhase (table:=ADR(phasesTable)):=		(phaseNumber:=3);
	//kran1Close:		ph_Kran (table:=ADR(phasesTable)):=			(phaseNumber:=4, Im:=Im.kran1, act:=DualStateImAction.off);
	//kran2Close:		ph_Kran (table:=ADR(phasesTable)):=			(phaseNumber:=5, Im:=Im.kran2, act:=DualStateImAction.off);
	P_zad:			CustomPhase (table:=ADR(phasesTable)):=		(phaseNumber:=6);
	kran5Open:		ph_Kran (table:=ADR(phasesTable)):=			(phaseNumber:=7, Im:=Im.kran5, act:=DualStateImAction.on);
	kran4Open:		ph_Kran (table:=ADR(phasesTable)):=			(phaseNumber:=8, Im:=Im.kran4, act:=DualStateImAction.on);
	kran5Close:		ph_Kran (table:=ADR(phasesTable)):=			(phaseNumber:=9, Im:=Im.kran5, act:=DualStateImAction.off);
	kran4Close:		ph_Kran (table:=ADR(phasesTable)):=			(phaseNumber:=10, Im:=Im.kran4, act:=DualStateImAction.off);
	{attribute 'symbol' := 'read'}
	timer10:		ph_Timer 	(table:=ADR(phasesTable)):=		(phaseNumber:=11, delay:=T#10S);
	P_vh_vyh_more_zad:	CustomPhase (table:=ADR(phasesTable)):=		(phaseNumber:=12);
	MaxZapolnenie_izm:REAL;
	Zapoln_Norm:	CustomPhase (table:=ADR(phasesTable)):=		(phaseNumber:=13);
	First_Step:		CustomPhase (table:=ADR(phasesTable)):=		(phaseNumber:=14);
END_VAR

SUPER^();
IF	algManager.mode <> ModeGpa.MODE_O THEN
	Opressovka_Start.ask ();
END_IF

IF	(Opressovka_Start.answer=Answers.ANS_YES) THEN
	Opressovka_Start.reset ();
	im.kran6.EnableOpcControl();
	algManager.setMode(nMode:=ModeGpa.MODE_O);
	OPC_Control.run();
	protections.p_DGazaNaVhodeNagnetatelja_GPA_STOP.reset ();
	protections.p_DGazaNaVyhodeNagnetatelja_GPA_STOP.reset ();
ELSIF	(Opressovka_Start.answer=Answers.ANS_no) THEN
		Opressovka_Start.reset ();
		reset ();
END_IF
/////////////////////////////////////////////////////
IF	OPC_Control.start AND NOT OPC_Control.top THEN
	PNS_NU_ON_Ask.ask ();
END_IF
IF	(PNS_NU_ON_Ask.answer=Answers.ANS_YES) AND NOT OPC_Control.top THEN
	OPC_Control.top:=TRUE;
	PNS_NU_ON_Ask.reset();
END_IF
IF	OPC_Control.top AND NOT Pms_more_50.start  THEN
	im.pns.EnableOpcControl();
	im.kran6.EnableOpcControl();
	Pms_more_50.run ();
	Pms_more_300.run ();
END_IF
IF	OPC_Control.top AND (im.pns.onStatus = statusDualInput.STATUS_On) AND NOT dPmg_more_100.start THEN
	im.nu.nu1.EnableOpcControl();
	im.nu.nu2.EnableOpcControl();
	dPmg_more_100.run ();
END_IF
/////////////////////////////////////////////////////
IF	((im.nu.nu1.onStatus = statusDualInput.STATUS_On) OR (im.nu.nu2.onStatus = statusDualInput.STATUS_On)) AND dPmg_more_100.start AND NOT dPmg_more_100.top THEN
	IF	((ai.PerepadDavlenieMasloGaz.interval	>=	statusAi.NORMAL) AND 
		(ai.PerepadDavlenieMasloGaz.value > 150)) AND (im.PerepadDavlenieMasloGaz_CK.status = 1) AND (NOT im.PerepadDavlenieMasloGaz_Less100.Q) THEN
		 dPmg_more_100.top:=TRUE;
		 protections.p_PerepadDavlenieMasloGaz.run ();
		 protections.p_PerepadDavlenieMasloGaz_Less100.run ();
	END_IF
END_IF
/////////////////////////////////////////////////////
IF	(im.pns.onStatus = statusDualInput.STATUS_On) AND Pms_more_50.start AND NOT Pms_more_50.top THEN
	IF	((ai.DavlenijaMasloSmNizkoe.interval	>=	statusAi.NORMAL) AND 
		(ai.DavlenijaMasloSmNizkoe.value > 50)) THEN
		 Pms_more_50.top:=TRUE;
		 protections.p_DavlenijaMasloSmNizkoe.run ();
	END_IF
END_IF
/////////////////////////////////////////////////////
IF	(im.pns.onStatus = statusDualInput.STATUS_On) AND Pms_more_300.start AND NOT Pms_more_300.top THEN
	IF	((ai.DavlenijaMasloSmVysokoe.interval	>=	statusAi.NORMAL) AND 
		(ai.DavlenijaMasloSmVysokoe.value > 300)) THEN
		 Pms_more_300.top:=TRUE;
		 protections.p_DavlenijaMasloSmVysokoe.run ();
	END_IF
END_IF
IF	dPmg_more_100.top AND Pms_more_50.top AND Pms_more_300.top THEN
	CASE	Auto.value OF
	0:	im.kran3.EnableOpcControl();
		im.kran4.EnableOpcControl();
		im.kran5.EnableOpcControl();
		im.kran3b.EnableOpcControl();
		Zapolnit_kontur.reset ();
		IF	im.PerepadDavlenieKran1_Less100.Q THEN
			im.kran1.EnableOpcControl();
			im.kran2.EnableOpcControl();
		ELSE
			im.kran1.DisableOpcControl();
			im.kran2.DisableOpcControl();
		END_IF
		P_vh_vyh_more_zad.reset ();
		kran5Open.reset ();
		kran4Open.reset ();
		timer10.reset ();
		kran5Close.reset ();
		P_zad.reset();
		First_Step.reset();
		kran4Close.reset ();
		MaxZapolnenie_izm:=0;
		MaxZapolnenie.setValue (0);
	1:	
		Zapoln_Norm.top:= (((MaxZapolnenie.value - MaxZapolnenie_izm) > 0.4) AND (MaxZapolnenie.value >= 0.4) AND (MaxZapolnenie.value <= 10) AND 
			(ai.DGazaNaVhodeNagnetatelja.interval >= statusAi.NORMAL) AND ((MaxZapolnenie.value - ai.DGazaNaVhodeNagnetatelja.value) > 0.4) AND 
			(ai.DGazaNaVyhodeNagnetatelja.interval >= statusAi.NORMAL) AND ((MaxZapolnenie.value - ai.DGazaNaVyhodeNagnetatelja.value) > 0.4 ));
		IF	(kran4Close.top AND Zapoln_Norm.top AND NOT P_zad.start) THEN
			P_vh_vyh_more_zad.reset ();
			kran5Open.reset ();
			kran4Open.reset ();
			timer10.reset ();
			kran5Close.reset ();
			kran4Close.reset ();
		END_IF
		IF	(NOT kran4Close.top) OR (kran4Close.top AND Zapoln_Norm.top AND NOT P_zad.start) THEN
		 	P_zad.run ();
			
		END_IF
		IF	(* NOT kran5Open.start AND*) (NOT P_zad.top) AND P_zad.start AND Zapoln_Norm.top THEN
			Zapolnit_kontur.ask ();
			im.kran3.DisableOpcControl();
			im.kran4.DisableOpcControl();
			im.kran5.DisableOpcControl();
			im.kran3b.DisableOpcControl();
			im.kran1.DisableOpcControl();
			im.kran2.DisableOpcControl();
			
			
		ELSIF	NOT Zapoln_Norm.top AND (NOT P_zad.top) THEN
				Zapolnit_kontur.reset ();
		END_IF
		IF	(Zapolnit_kontur.answer=Answers.ANS_YES) AND P_zad.start THEN
			MaxZapolnenie_izm:= MaxZapolnenie.value;
			IF 	NOT First_Step.top THEN
				kran5Open.run ();
			ELSE
				kran4Open.run ();
			END_IF
			Zapolnit_kontur.reset ();
			P_zad.top:=TRUE;
		END_IF
		IF	P_zad.top AND NOT kran4Close.top THEN
			MaxZapolnenie.newvalue:=MaxZapolnenie_izm;
		ELSE
			MaxZapolnenie.newvalue:= MaxZapolnenie.newvalue; 
		END_IF;
		IF	kran5Open.top AND NOT (First_Step.top) THEN
			kran4Open.run ();
		END_IF;
		IF 	kran4Open.top AND NOT timer10.top AND NOT (First_Step.top) THEN
			timer10.run ();
		END_IF;
		IF	timer10.top AND NOT (First_Step.top) THEN
			kran5Close.run ();
		END_IF
		IF	(kran5Close.top) OR (First_Step.top AND kran4Open.top) THEN
			P_vh_vyh_more_zad.run ();
		END_IF
		IF	(ai.DGazaNaVhodeNagnetatelja.interval >= statusAi.NORMAL) AND (ai.DGazaNaVhodeNagnetatelja.value >= MaxZapolnenie.value) AND 
			(ai.DGazaNaVyhodeNagnetatelja.interval >= statusAi.NORMAL) AND (ai.DGazaNaVyhodeNagnetatelja.value >= MaxZapolnenie.value)AND  P_vh_vyh_more_zad.start AND NOT P_vh_vyh_more_zad.top THEN
			kran4Close.run();
			P_vh_vyh_more_zad.top:=TRUE;
		END_IF;
		IF	kran4Close.top THEN
			First_Step.top:=TRUE;
			im.kran3.EnableOpcControl();
			im.kran4.EnableOpcControl();
			im.kran5.EnableOpcControl();
			im.kran3b.EnableOpcControl();
			IF	Zapoln_Norm.top THEN
				P_zad.reset();
			END_IF
			IF	im.PerepadDavlenieKran1_less100.Q THEN
				im.kran1.EnableOpcControl();
				im.kran2.EnableOpcControl();	
			ELSE
				im.kran1.DisableOpcControl();
				im.kran2.DisableOpcControl();
			END_IF
		ELSE
			im.kran1.DisableOpcControl();
			im.kran2.DisableOpcControl();
		END_IF
	END_CASE
END_IF

METHOD PUBLIC reset
VAR_INPUT
END_VAR
SUPER^.reset();
Auto.setValue (0);
Opressovka_Start.reset ();
MaxZapolnenie.setValue (0);
statusSet.setBit(15,0);
im.kran6.DisableOpcControl();
im.kran1.DisableOpcControl();
im.kran2.DisableOpcControl();
im.kran3.DisableOpcControl();
im.kran4.DisableOpcControl();
im.kran5.DisableOpcControl();
im.kran3b.DisableOpcControl();
im.pns.DisableOpcControl();
im.nu.nu1.DisableOpcControl();
im.nu.nu2.DisableOpcControl();
PNS_NU_ON_Ask.reset();
Zapolnit_kontur.reset ();
MaxZapolnenie_izm:=0;
END_METHOD

END_FUNCTION_BLOCK

// K2/std12k5/Prov/Opressovka
{attribute 'symbol' := 'none'}
FUNCTION_BLOCK Opressovka EXTENDS StepBySteapAlgoritm
VAR_INPUT
	{attribute 'symbol' := 'read'}
	Auto:DiscretParametr(table:=ADR(objectTable));//{name:Автоматический или ручной режим работы}
	{attribute 'symbol' := 'read'}
	MaxZapolnenie:AnalogParametr(table:=ADR(objectTable));//{name:задайте сюда значение}
END_VAR
VAR_OUTPUT
	{attribute 'symbol' := 'read'}
	Opressovka_Start:		Question(table:=ADR(ObjectTable)):=			(AnswerVariants:=(Answers.ANS_YES OR Answers.ANS_NO));
	{attribute 'symbol' := 'read'}
	PNS_NU_ON_Ask:		Question(table:=ADR(ObjectTable)):=			(AnswerVariants:=Answers.ANS_YES);
	{attribute 'symbol' := 'read'}
	Zapolnit_kontur:	Question(table:=ADR(ObjectTable)):=			(AnswerVariants:=Answers.ANS_YES);
END_VAR
VAR
	OPC_Control:	CustomPhase (table:=ADR(phasesTable)):=		(phaseNumber:=0);
	Pms_more_50:	CustomPhase (table:=ADR(phasesTable)):=		(phaseNumber:=1);
	Pms_more_300:	CustomPhase (table:=ADR(phasesTable)):=		(phaseNumber:=2);
	dPmg_more_100:	CustomPhase (table:=ADR(phasesTable)):=		(phaseNumber:=3);
	//kran1Close:		ph_Kran (table:=ADR(phasesTable)):=			(phaseNumber:=4, Im:=Im.kran1, act:=DualStateImAction.off);
	//kran2Close:		ph_Kran (table:=ADR(phasesTable)):=			(phaseNumber:=5, Im:=Im.kran2, act:=DualStateImAction.off);
	P_zad:			CustomPhase (table:=ADR(phasesTable)):=		(phaseNumber:=6);
	kran5Open:		ph_Kran (table:=ADR(phasesTable)):=			(phaseNumber:=7, Im:=Im.kran5, act:=DualStateImAction.on);
	kran4Open:		ph_Kran (table:=ADR(phasesTable)):=			(phaseNumber:=8, Im:=Im.kran4, act:=DualStateImAction.on);
	kran5Close:		ph_Kran (table:=ADR(phasesTable)):=			(phaseNumber:=9, Im:=Im.kran5, act:=DualStateImAction.off);
	kran4Close:		ph_Kran (table:=ADR(phasesTable)):=			(phaseNumber:=10, Im:=Im.kran4, act:=DualStateImAction.off);
	{attribute 'symbol' := 'read'}
	timer10:		ph_Timer 	(table:=ADR(phasesTable)):=		(phaseNumber:=11, delay:=T#10S);
	P_vh_vyh_more_zad:	CustomPhase (table:=ADR(phasesTable)):=		(phaseNumber:=12);
	MaxZapolnenie_izm:REAL;
	Zapoln_Norm:	CustomPhase (table:=ADR(phasesTable)):=		(phaseNumber:=13);
	First_Step:		CustomPhase (table:=ADR(phasesTable)):=		(phaseNumber:=14);
END_VAR

SUPER^();
IF	algManager.mode <> ModeGpa.MODE_O THEN
	Opressovka_Start.ask ();
END_IF

IF	(Opressovka_Start.answer=Answers.ANS_YES) THEN
	Opressovka_Start.reset ();
	im.kran6.EnableOpcControl();
	algManager.setMode(nMode:=ModeGpa.MODE_O);
	OPC_Control.run();
	protections.p_DGazaNaVhodeNagnetatelja_GPA_STOP.reset ();
	protections.p_DGazaNaVyhodeNagnetatelja_GPA_STOP.reset ();
ELSIF	(Opressovka_Start.answer=Answers.ANS_no) THEN
		Opressovka_Start.reset ();
		reset ();
END_IF
/////////////////////////////////////////////////////
IF	OPC_Control.start AND NOT OPC_Control.top THEN
	PNS_NU_ON_Ask.ask ();
END_IF
IF	(PNS_NU_ON_Ask.answer=Answers.ANS_YES) AND NOT OPC_Control.top THEN
	OPC_Control.top:=TRUE;
	PNS_NU_ON_Ask.reset();
END_IF
IF	OPC_Control.top AND NOT Pms_more_50.start  THEN
	im.pns.EnableOpcControl();
	im.kran6.EnableOpcControl();
	Pms_more_50.run ();
	Pms_more_300.run ();
END_IF
IF	OPC_Control.top AND (im.pns.onStatus = statusDualInput.STATUS_On) AND NOT dPmg_more_100.start THEN
	im.nu.nu1.EnableOpcControl();
	im.nu.nu2.EnableOpcControl();
	dPmg_more_100.run ();
END_IF
/////////////////////////////////////////////////////
IF	((im.nu.nu1.onStatus = statusDualInput.STATUS_On) OR (im.nu.nu2.onStatus = statusDualInput.STATUS_On)) AND dPmg_more_100.start AND NOT dPmg_more_100.top THEN
	IF	((ai.PerepadDavlenieMasloGaz.interval	>=	statusAi.NORMAL) AND 
		(ai.PerepadDavlenieMasloGaz.value > 150)) AND (im.PerepadDavlenieMasloGaz_CK.status = 1) AND (NOT im.PerepadDavlenieMasloGaz_Less100.Q) THEN
		 dPmg_more_100.top:=TRUE;
		 protections.p_PerepadDavlenieMasloGaz.run ();
		 protections.p_PerepadDavlenieMasloGaz_Less100.run ();
	END_IF
END_IF
/////////////////////////////////////////////////////
IF	(im.pns.onStatus = statusDualInput.STATUS_On) AND Pms_more_50.start AND NOT Pms_more_50.top THEN
	IF	((ai.DavlenijaMasloSmNizkoe.interval	>=	statusAi.NORMAL) AND 
		(ai.DavlenijaMasloSmNizkoe.value > 50)) THEN
		 Pms_more_50.top:=TRUE;
		 protections.p_DavlenijaMasloSmNizkoe.run ();
	END_IF
END_IF
/////////////////////////////////////////////////////
IF	(im.pns.onStatus = statusDualInput.STATUS_On) AND Pms_more_300.start AND NOT Pms_more_300.top THEN
	IF	((ai.DavlenijaMasloSmVysokoe.interval	>=	statusAi.NORMAL) AND 
		(ai.DavlenijaMasloSmVysokoe.value > 300)) THEN
		 Pms_more_300.top:=TRUE;
		 protections.p_DavlenijaMasloSmVysokoe.run ();
	END_IF
END_IF
IF	dPmg_more_100.top AND Pms_more_50.top AND Pms_more_300.top THEN
	CASE	Auto.value OF
	0:	im.kran3.EnableOpcControl();
		im.kran4.EnableOpcControl();
		im.kran5.EnableOpcControl();
		im.kran3b.EnableOpcControl();
		Zapolnit_kontur.reset ();
		IF	im.PerepadDavlenieKran1_Less100.Q THEN
			im.kran1.EnableOpcControl();
			im.kran2.EnableOpcControl();
		ELSE
			im.kran1.DisableOpcControl();
			im.kran2.DisableOpcControl();
		END_IF
		P_vh_vyh_more_zad.reset ();
		kran5Open.reset ();
		kran4Open.reset ();
		timer10.reset ();
		kran5Close.reset ();
		P_zad.reset();
		First_Step.reset();
		kran4Close.reset ();
		MaxZapolnenie_izm:=0;
		MaxZapolnenie.setValue (0);
	1:	
		Zapoln_Norm.top:= (((MaxZapolnenie.value - MaxZapolnenie_izm) > 0.4) AND (MaxZapolnenie.value >= 0.4) AND (MaxZapolnenie.value <= 10) AND 
			(ai.DGazaNaVhodeNagnetatelja.interval >= statusAi.NORMAL) AND ((MaxZapolnenie.value - ai.DGazaNaVhodeNagnetatelja.value) > 0.4) AND 
			(ai.DGazaNaVyhodeNagnetatelja.interval >= statusAi.NORMAL) AND ((MaxZapolnenie.value - ai.DGazaNaVyhodeNagnetatelja.value) > 0.4 ));
		IF	(kran4Close.top AND Zapoln_Norm.top AND NOT P_zad.start) THEN
			P_vh_vyh_more_zad.reset ();
			kran5Open.reset ();
			kran4Open.reset ();
			timer10.reset ();
			kran5Close.reset ();
			kran4Close.reset ();
		END_IF
		IF	(NOT kran4Close.top) OR (kran4Close.top AND Zapoln_Norm.top AND NOT P_zad.start) THEN
		 	P_zad.run ();
			
		END_IF
		IF	(* NOT kran5Open.start AND*) (NOT P_zad.top) AND P_zad.start AND Zapoln_Norm.top THEN
			Zapolnit_kontur.ask ();
			im.kran3.DisableOpcControl();
			im.kran4.DisableOpcControl();
			im.kran5.DisableOpcControl();
			im.kran3b.DisableOpcControl();
			im.kran1.DisableOpcControl();
			im.kran2.DisableOpcControl();
			
			
		ELSIF	NOT Zapoln_Norm.top AND (NOT P_zad.top) THEN
				Zapolnit_kontur.reset ();
		END_IF
		IF	(Zapolnit_kontur.answer=Answers.ANS_YES) AND P_zad.start THEN
			MaxZapolnenie_izm:= MaxZapolnenie.value;
			IF 	NOT First_Step.top THEN
				kran5Open.run ();
			ELSE
				kran4Open.run ();
			END_IF
			Zapolnit_kontur.reset ();
			P_zad.top:=TRUE;
		END_IF
		IF	P_zad.top AND NOT kran4Close.top THEN
			MaxZapolnenie.newvalue:=MaxZapolnenie_izm;
		ELSE
			MaxZapolnenie.newvalue:= MaxZapolnenie.newvalue; 
		END_IF;
		IF	kran5Open.top AND NOT (First_Step.top) THEN
			kran4Open.run ();
		END_IF;
		IF 	kran4Open.top AND NOT timer10.top AND NOT (First_Step.top) THEN
			timer10.run ();
		END_IF;
		IF	timer10.top AND NOT (First_Step.top) THEN
			kran5Close.run ();
		END_IF
		IF	(kran5Close.top) OR (First_Step.top AND kran4Open.top) THEN
			P_vh_vyh_more_zad.run ();
		END_IF
		IF	(ai.DGazaNaVhodeNagnetatelja.interval >= statusAi.NORMAL) AND (ai.DGazaNaVhodeNagnetatelja.value >= MaxZapolnenie.value) AND 
			(ai.DGazaNaVyhodeNagnetatelja.interval >= statusAi.NORMAL) AND (ai.DGazaNaVyhodeNagnetatelja.value >= MaxZapolnenie.value)AND  P_vh_vyh_more_zad.start AND NOT P_vh_vyh_more_zad.top THEN
			kran4Close.run();
			P_vh_vyh_more_zad.top:=TRUE;
		END_IF;
		IF	kran4Close.top THEN
			First_Step.top:=TRUE;
			im.kran3.EnableOpcControl();
			im.kran4.EnableOpcControl();
			im.kran5.EnableOpcControl();
			im.kran3b.EnableOpcControl();
			IF	Zapoln_Norm.top THEN
				P_zad.reset();
			END_IF
			IF	im.PerepadDavlenieKran1_less100.Q THEN
				im.kran1.EnableOpcControl();
				im.kran2.EnableOpcControl();	
			ELSE
				im.kran1.DisableOpcControl();
				im.kran2.DisableOpcControl();
			END_IF
		ELSE
			im.kran1.DisableOpcControl();
			im.kran2.DisableOpcControl();
		END_IF
	END_CASE
END_IF

METHOD PUBLIC reset
VAR_INPUT
END_VAR
SUPER^.reset();
Auto.setValue (0);
Opressovka_Start.reset ();
MaxZapolnenie.setValue (0);
statusSet.setBit(15,0);
im.kran6.DisableOpcControl();
im.kran1.DisableOpcControl();
im.kran2.DisableOpcControl();
im.kran3.DisableOpcControl();
im.kran4.DisableOpcControl();
im.kran5.DisableOpcControl();
im.kran3b.DisableOpcControl();
im.pns.DisableOpcControl();
im.nu.nu1.DisableOpcControl();
im.nu.nu2.DisableOpcControl();
PNS_NU_ON_Ask.reset();
Zapolnit_kontur.reset ();
MaxZapolnenie_izm:=0;
END_METHOD

END_FUNCTION_BLOCK

// K1/std12k5/Prov/Prov_dPmg
{attribute 'symbol' := 'none'}
FUNCTION_BLOCK Prov_dPmg EXTENDS StepBySteapAlgoritm
VAR_INPUT
END_VAR
VAR_OUTPUT
	{attribute 'symbol' := 'read'}
	NU_OFF_Ask:		Question(table:=ADR(ObjectTable)):=			(AnswerVariants:=Answers.ANS_YES);
END_VAR
VAR
	nuOff:			ph_Switch 	(table:=ADR(phasesTable)):=		(phaseNumber:=0, Im:=Im.nu, act:=DualStateImAction.off);
	pnsOff:			ph_Switch 	(table:=ADR(phasesTable)):=		(phaseNumber:=1, Im:=Im.pns, act:=DualStateImAction.off);
	{attribute 'symbol' := 'read'}
	timer120:		ph_Timer 	(table:=ADR(phasesTable)):=		(phaseNumber:=2, delay:=T#120S);
	dPmg_less_100:	CustomPhase (table:=ADR(phasesTable)):=		(phaseNumber:=3);
	nuOn:			CustomPhase (table:=ADR(phasesTable)):=		(phaseNumber:=4);
	pnsOn:			ph_Switch 	(table:=ADR(phasesTable)):=		(phaseNumber:=5, Im:=Im.pns, act:=DualStateImAction.on);
	Error_Alg: 		CustomPhase (table:=ADR(phasesTable)):=		(phaseNumber:=6);
	dPmg_more_100:	CustomPhase (table:=ADR(phasesTable)):=		(phaseNumber:=7);
END_VAR

SUPER^();
IF	NOT nuOff.start THEN
	NU_OFF_Ask.ask ();
END_IF;
IF	(nu_OFF_Ask.answer=Answers.ANS_YES) THEN
	nuOff.run (); //Отключаем НУ
	pnsOff.run ();
	NU_OFF_Ask.reset ();
	timer120.run (); //Запускаем таймер 120 секунд
END_IF

/////////////////////////////////////////
IF	nuOff.top THEN  //запуск фазы на давление меньше 100
	dPmg_less_100.run ();
END_IF
/////////////////////////////////////////
IF	dPmg_less_100.start AND (NOT dPmg_less_100.top) THEN //Перепад маслогаз меньше 100 по аналогу и дискрету
	IF 	im.PerepadDavlenieMasloGaz_Less100.Q AND (ai.PerepadDavlenieMasloGaz.value < 150) THEN
	  	dPmg_less_100.top:=TRUE;
		nuOn.run ();
		pnsOn.run ();
	END_IF
END_IF

/////////////////////////////////////////
IF	((im.nu.nu1.onStatus = statusDualInput.STATUS_ON) OR (im.nu.nu2.onStatus = statusDualInput.STATUS_ON))  AND nuOn.start  AND NOT nuOn.top THEN
	nuOn.top := TRUE;
END_IF
/////////////////////////////////////////
IF	timer120.top THEN //Ошибка завершения алгоритма по таймеру
	Error_Alg.ERROR := TRUE;
ELSE
	Error_Alg.ERROR := FALSE;	
END_IF
/////////////////////////////////////////
IF	nuOn.top AND pnsOn.top THEN //если насос переключился, то завершаем алгоритм
	dPmg_more_100.run ();
END_IF
/////////////////////////////////////////
IF	dPmg_more_100.start AND (NOT dPmg_more_100.top) AND NOT (algoritms.autoNu_1.flag1 OR algoritms.autoNu_1.flag2) THEN //Перепад маслогаз больше 100 по аналогу и дискрету
	IF 	(NOT im.PerepadDavlenieMasloGaz_Less100.Q) AND (im.PerepadDavlenieMasloGaz_CK.status = 1) AND  (ai.PerepadDavlenieMasloGaz.value > 150) THEN
		dPmg_more_100.top :=TRUE;
		timer120.reset ();
		end ();
	END_IF
END_IF

METHOD PUBLIC reset
VAR_INPUT
END_VAR
SUPER^.reset();
statusSet.setBit(15,0);
NU_OFF_Ask.reset ();
END_METHOD

METHOD PUBLIC run
VAR_INPUT
END_VAR
SUPER^.run();
statusSet.setBit(15,1);
protections.p_DavlenijaMasloSmNizkoe.reset ();
protections.p_DavlenijaMasloSmVysokoe.reset ();
END_METHOD

END_FUNCTION_BLOCK

// K2/std12k5/Prov/Prov_dPmg
{attribute 'symbol' := 'none'}
FUNCTION_BLOCK Prov_dPmg EXTENDS StepBySteapAlgoritm
VAR_INPUT
END_VAR
VAR_OUTPUT
	{attribute 'symbol' := 'read'}
	NU_OFF_Ask:		Question(table:=ADR(ObjectTable)):=			(AnswerVariants:=Answers.ANS_YES);
END_VAR
VAR
	nuOff:			ph_Switch 	(table:=ADR(phasesTable)):=		(phaseNumber:=0, Im:=Im.nu, act:=DualStateImAction.off);
	pnsOff:			ph_Switch 	(table:=ADR(phasesTable)):=		(phaseNumber:=1, Im:=Im.pns, act:=DualStateImAction.off);
	{attribute 'symbol' := 'read'}
	timer120:		ph_Timer 	(table:=ADR(phasesTable)):=		(phaseNumber:=2, delay:=T#120S);
	dPmg_less_100:	CustomPhase (table:=ADR(phasesTable)):=		(phaseNumber:=3);
	nuOn:			CustomPhase (table:=ADR(phasesTable)):=		(phaseNumber:=4);
	pnsOn:			ph_Switch 	(table:=ADR(phasesTable)):=		(phaseNumber:=5, Im:=Im.pns, act:=DualStateImAction.on);
	Error_Alg: 		CustomPhase (table:=ADR(phasesTable)):=		(phaseNumber:=6);
	dPmg_more_100:	CustomPhase (table:=ADR(phasesTable)):=		(phaseNumber:=7);
END_VAR

SUPER^();
IF	NOT nuOff.start THEN
	NU_OFF_Ask.ask ();
END_IF;
IF	(nu_OFF_Ask.answer=Answers.ANS_YES) THEN
	nuOff.run (); //Отключаем НУ
	pnsOff.run ();
	NU_OFF_Ask.reset ();
	timer120.run (); //Запускаем таймер 120 секунд
END_IF

/////////////////////////////////////////
IF	nuOff.top THEN  //запуск фазы на давление меньше 100
	dPmg_less_100.run ();
END_IF
/////////////////////////////////////////
IF	dPmg_less_100.start AND (NOT dPmg_less_100.top) THEN //Перепад маслогаз меньше 100 по аналогу и дискрету
	IF 	im.PerepadDavlenieMasloGaz_Less100.Q AND (ai.PerepadDavlenieMasloGaz.value < 150) THEN
	  	dPmg_less_100.top:=TRUE;
		nuOn.run ();
		pnsOn.run ();
	END_IF
END_IF

/////////////////////////////////////////
IF	((im.nu.nu1.onStatus = statusDualInput.STATUS_ON) OR (im.nu.nu2.onStatus = statusDualInput.STATUS_ON))  AND nuOn.start  AND NOT nuOn.top THEN
	nuOn.top := TRUE;
END_IF
/////////////////////////////////////////
IF	timer120.top THEN //Ошибка завершения алгоритма по таймеру
	Error_Alg.ERROR := TRUE;
ELSE
	Error_Alg.ERROR := FALSE;	
END_IF
/////////////////////////////////////////
IF	nuOn.top AND pnsOn.top THEN //если насос переключился, то завершаем алгоритм
	dPmg_more_100.run ();
END_IF
/////////////////////////////////////////
IF	dPmg_more_100.start AND (NOT dPmg_more_100.top) AND NOT (algoritms.autoNu_1.flag1 OR algoritms.autoNu_1.flag2) THEN //Перепад маслогаз больше 100 по аналогу и дискрету
	IF 	(NOT im.PerepadDavlenieMasloGaz_Less100.Q) AND (im.PerepadDavlenieMasloGaz_CK.status = 1) AND  (ai.PerepadDavlenieMasloGaz.value > 150) THEN
		dPmg_more_100.top :=TRUE;
		timer120.reset ();
		end ();
	END_IF
END_IF

METHOD PUBLIC reset
VAR_INPUT
END_VAR
SUPER^.reset();
statusSet.setBit(15,0);
NU_OFF_Ask.reset ();
END_METHOD

METHOD PUBLIC run
VAR_INPUT
END_VAR
SUPER^.run();
statusSet.setBit(15,1);
protections.p_DavlenijaMasloSmNizkoe.reset ();
protections.p_DavlenijaMasloSmVysokoe.reset ();
END_METHOD

END_FUNCTION_BLOCK

// K1/std12k5/Prov/Prov_Pms
{attribute 'symbol' := 'none'}
FUNCTION_BLOCK Prov_Pms EXTENDS StepBySteapAlgoritm
VAR_INPUT
END_VAR
VAR_OUTPUT
	{attribute 'symbol' := 'read'}
	PNS_OFF_Ask:		Question(table:=ADR(ObjectTable)):=			(AnswerVariants:=Answers.ANS_YES);
END_VAR
VAR
	
	pnsOff:			ph_Switch 	(table:=ADR(phasesTable)):=		(phaseNumber:=0, Im:=Im.pns, act:=DualStateImAction.off);
	{attribute 'symbol' := 'read'}
	timer120:		ph_Timer 	(table:=ADR(phasesTable)):=		(phaseNumber:=1, delay:=T#120S);
	Pms_less_25:	CustomPhase (table:=ADR(phasesTable)):=		(phaseNumber:=2);
	Pms_less_250:	CustomPhase (table:=ADR(phasesTable)):=		(phaseNumber:=3);
	Error_Alg: 		CustomPhase (table:=ADR(phasesTable)):=		(phaseNumber:=4);
END_VAR

SUPER^();
IF	NOT pnsOff.start THEN
	PNS_OFF_Ask.ask ();
END_IF
IF	(PNS_OFF_Ask.answer=Answers.ANS_YES) THEN
	pnsOff.run (); //отключаем ПНС
	PNS_OFF_Ask.reset ();
	IF	NOT (Pms_less_250.top AND Pms_less_25.top) THEN
		timer120.run (); //запускаем таймер 120 секунд
	END_IF
END_IF

/////////////////////////////////////////
IF	pnsOff.top  THEN //запускаем фазу на проверку давления маслосмазки
	Pms_less_25.run ();
	Pms_less_250.run ();
END_IF
/////////////////////////////////////////
IF	Pms_less_25.start AND (NOT Pms_less_25.top) THEN //Давление маслосмазки низкое меньше 25 кПа
	IF 	(ai.DavlenijaMasloSmNizkoe.interval>=statusAi.NORMAL) AND (ai.DavlenijaMasloSmNizkoe.value < 25) THEN
	  	Pms_less_25.top:=TRUE;
	END_IF
END_IF
/////////////////////////////////////////
IF	Pms_less_250.start AND (NOT Pms_less_250.top) THEN //Давление маслосмазки высокое меньше 250 кПа
	IF	(ai.DavlenijaMasloSmVysokoe.interval>=statusAi.NORMAL) AND (ai.DavlenijaMasloSmVysokoe.value < 250) THEN
	  	Pms_less_250.top:=TRUE;
	END_IF
END_IF
/////////////////////////////////////////
IF	timer120.top THEN //Ошибка завершения алгоритма по таймеру
	Error_Alg.ERROR := TRUE;
ELSE
	Error_Alg.ERROR := FALSE;	
END_IF
/////////////////////////////////////////
IF	Pms_less_250.top AND Pms_less_25.top  THEN //если давление упало по дискрету и аналогу завершаем алгоритм
	timer120.reset ();
	end ();
END_IF

METHOD PUBLIC reset
VAR_INPUT
END_VAR
SUPER^.reset();
statusSet.setBit(15,0);
PNS_OFF_Ask.reset ();
END_METHOD

METHOD PUBLIC run
VAR_INPUT
END_VAR
SUPER^.run();
statusSet.setBit(15,1);
END_METHOD

END_FUNCTION_BLOCK

// K2/std12k5/Prov/Prov_Pms
{attribute 'symbol' := 'none'}
FUNCTION_BLOCK Prov_Pms EXTENDS StepBySteapAlgoritm
VAR_INPUT
END_VAR
VAR_OUTPUT
	{attribute 'symbol' := 'read'}
	PNS_OFF_Ask:		Question(table:=ADR(ObjectTable)):=			(AnswerVariants:=Answers.ANS_YES);
END_VAR
VAR
	
	pnsOff:			ph_Switch 	(table:=ADR(phasesTable)):=		(phaseNumber:=0, Im:=Im.pns, act:=DualStateImAction.off);
	{attribute 'symbol' := 'read'}
	timer120:		ph_Timer 	(table:=ADR(phasesTable)):=		(phaseNumber:=1, delay:=T#120S);
	Pms_less_25:	CustomPhase (table:=ADR(phasesTable)):=		(phaseNumber:=2);
	Pms_less_250:	CustomPhase (table:=ADR(phasesTable)):=		(phaseNumber:=3);
	Error_Alg: 		CustomPhase (table:=ADR(phasesTable)):=		(phaseNumber:=4);
END_VAR

SUPER^();
IF	NOT pnsOff.start THEN
	PNS_OFF_Ask.ask ();
END_IF
IF	(PNS_OFF_Ask.answer=Answers.ANS_YES) THEN
	pnsOff.run (); //отключаем ПНС
	PNS_OFF_Ask.reset ();
	IF	NOT (Pms_less_250.top AND Pms_less_25.top) THEN
		timer120.run (); //запускаем таймер 120 секунд
	END_IF
END_IF

/////////////////////////////////////////
IF	pnsOff.top  THEN //запускаем фазу на проверку давления маслосмазки
	Pms_less_25.run ();
	Pms_less_250.run ();
END_IF
/////////////////////////////////////////
IF	Pms_less_25.start AND (NOT Pms_less_25.top) THEN //Давление маслосмазки низкое меньше 25 кПа
	IF 	(ai.DavlenijaMasloSmNizkoe.interval>=statusAi.NORMAL) AND (ai.DavlenijaMasloSmNizkoe.value < 25) THEN
	  	Pms_less_25.top:=TRUE;
	END_IF
END_IF
/////////////////////////////////////////
IF	Pms_less_250.start AND (NOT Pms_less_250.top) THEN //Давление маслосмазки высокое меньше 250 кПа
	IF	(ai.DavlenijaMasloSmVysokoe.interval>=statusAi.NORMAL) AND (ai.DavlenijaMasloSmVysokoe.value < 250) THEN
	  	Pms_less_250.top:=TRUE;
	END_IF
END_IF
/////////////////////////////////////////
IF	timer120.top THEN //Ошибка завершения алгоритма по таймеру
	Error_Alg.ERROR := TRUE;
ELSE
	Error_Alg.ERROR := FALSE;	
END_IF
/////////////////////////////////////////
IF	Pms_less_250.top AND Pms_less_25.top  THEN //если давление упало по дискрету и аналогу завершаем алгоритм
	timer120.reset ();
	end ();
END_IF

METHOD PUBLIC reset
VAR_INPUT
END_VAR
SUPER^.reset();
statusSet.setBit(15,0);
PNS_OFF_Ask.reset ();
END_METHOD

METHOD PUBLIC run
VAR_INPUT
END_VAR
SUPER^.run();
statusSet.setBit(15,1);
END_METHOD

END_FUNCTION_BLOCK

// K1/std12k5/Pusk/ppuAlg
	{attribute 'symbol' := 'none'}
FUNCTION_BLOCK ppuAlg EXTENDS StepBySteapAlgoritm
VAR_INPUT
END_VAR
VAR_OUTPUT
	{attribute 'symbol' := 'read'}
	ppuFirst_for_Pusk_Ch:BOOL;
	{attribute 'symbol' := 'read'}
	ppuFirst_for_Pusk_R:BOOL;
	{attribute 'symbol' := 'read'}
	ppuFirst_for_V_Ch:BOOL;
	{attribute 'symbol' := 'read'}
	ppuFirst_for_V_R:BOOL;
	{attribute 'symbol' := 'read'}
	ppuFirst_for_Pms_dPmg: BOOL;
	{attribute 'symbol' := 'read'}
	ppuFirst_for_K: BOOL;
	{attribute 'symbol' := 'read'}
	ppuFirst_for_I: BOOL;
	{attribute 'symbol' := 'read'}
	ppuSecond_V_Pusk_Ch: BOOL;
	{attribute 'symbol' := 'read'}
	ppuSecond_V_Pusk_R: BOOL;
	{attribute 'symbol' := 'read'}
	ppuSecond_I: BOOL;
	{attribute 'symbol' := 'read'}
	ppuThird:BOOL;
	{attribute 'symbol' := 'read'}
	ppuForth:BOOL;
END_VAR
VAR
	BMP_Err:					CustomPhase (table:=ADR(phasesTable)):=		(phaseNumber:=0); //Все аналоги исправны
	
	Level_masla_Norm: 			CustomPhase (table:=ADR(phasesTable)):=		(phaseNumber:=1); //уровень масла в МЮ нормальный
	
	T_masla_Norm: 				CustomPhase (table:=ADR(phasesTable)):=		(phaseNumber:=2); //температура масла в мб больше 25
	
	Krans_ready_to_move:		CustomPhase (table:=ADR(phasesTable)):=		(phaseNumber:=3); //Краны готовы к управлению
	
	Krans_Poloj:				CustomPhase (table:=ADR(phasesTable)):=		(phaseNumber:=4); //Положение кранов соответствует ППУ
	
	Net_AO_KC_SHKS04M: 			CustomPhase (table:=ADR(phasesTable)):=		(phaseNumber:=5); //Нет АО от ШКС
	
	EGPA_Stop:					CustomPhase (table:=ADR(phasesTable)):=		(phaseNumber:=6); //ЭГПА остановлен
	
	Avt_SHU_vkl:				CustomPhase (table:=ADR(phasesTable)):=		(phaseNumber:=7); //Автомат в ячейке ШУ включен
	
	All_IM_Off:					CustomPhase (table:=ADR(phasesTable)):=		(phaseNumber:=8); //Все ИМ выключены
	
	Nalichie220_SHU_Ai:			CustomPhase (table:=ADR(phasesTable)):=		(phaseNumber:=9); //Напряжение в ШУ в норме по AI
	
	BP_Norm:					CustomPhase (table:=ADR(phasesTable)):=		(phaseNumber:=10); //Все БП исправны
	
	Naprajenie_U_IM: 			CustomPhase (table:=ADR(phasesTable)):=		(phaseNumber:=11); //есть напряжение в цепях управления ИМ
	
	MV_Poloj_RolledON:			CustomPhase (table:=ADR(phasesTable)):=		(phaseNumber:=12); //Тележка МВ вкачена
	
	MV_Poloj_RolledOFF:			CustomPhase (table:=ADR(phasesTable)):=		(phaseNumber:=13); //Тележка МВ выкачена 
	
	NOTAnalogNS: 				CustomPhase (table:=ADR(phasesTable)):=		(phaseNumber:=14); //Все аналоги исправны
	
	Net_ASPS_Analogs:			CustomPhase (table:=ADR(phasesTable)):=		(phaseNumber:=15); //Нет АС и ПС по аналогам
	
	Not_AS:						CustomPhase (table:=ADR(phasesTable)):=		(phaseNumber:=16); //Нет сработанных защит
	
	Gotov_Vozb:					CustomPhase (table:=ADR(phasesTable)):=		(phaseNumber:=17); //Возбудитель Готов
	
	Reactornyi_P:				CustomPhase (table:=ADR(phasesTable)):=		(phaseNumber:=18); //Реакторный пуск
	
	Chastotnyi_P:				CustomPhase (table:=ADR(phasesTable)):=		(phaseNumber:=19); //Частотный пуск
	
	dP_kr1:						CustomPhase (table:=ADR(phasesTable)):=		(phaseNumber:=20); //Перепад на кране один есть
	
	Auto_Rej:					CustomPhase (table:=ADR(phasesTable)):=		(phaseNumber:=21); //ПНС, НУ в автоматическом режиме
	
	CK_IM_Norm: 				CustomPhase (table:=ADR(phasesTable)):=		(phaseNumber:=22); //Цепи контроля ИМ исправны
	
	HAnd_Mode:					CustomPhase (table:=ADR(phasesTable)):=		(phaseNumber:=23); //Ручной режим
	
	Impuls_Gaz:					CustomPhase (table:=ADR(phasesTable)):=		(phaseNumber:=24); //импульсный газ	
	
END_VAR

SUPER^();
BMP_Err.top:= ((BMPERR_k = 0) OR (kontroller.imit));
/////////////////////////////////////////
Level_masla_Norm.top:=(ai.YrovenMaslaMB.interval=statusAi.normal);//уровень масла в норме
/////////////////////////////////////////
T_masla_Norm.top:=(ai.TMaslaMB.interval=statusAi.normal);//температура масла в норме
/////////////////////////////////////////
Krans_ready_to_move.top:= 	NOT (im.kran1.so OR im.kran1.sz OR im.kran2.so OR im.kran2.sz OR im.kran3.so OR im.kran3.sz OR im.kran3b.so OR im.kran3b.sz OR im.kran4.so OR im.kran4.sz OR
							im.kran5.so OR im.kran5.sz OR im.kran6.so OR im.kran6.sz); //Краны готовы к управлению
/////////////////////////////////////////
Krans_Poloj.top:=		(Im.kran1.onStatus=statusDualInput.STATUS_OFF) AND
						(Im.kran2.onStatus=statusDualInput.STATUS_OFF) AND
						(Im.kran3.onStatus=statusDualInput.STATUS_OFF) AND
						(Im.kran3b.onStatus=statusDualInput.STATUS_ON) AND
						(Im.kran4.onStatus=statusDualInput.STATUS_OFF) AND
						(Im.kran5.onStatus=statusDualInput.STATUS_ON) AND 
						(Im.kran6.onStatus=statusDualInput.STATUS_ON); 
/////////////////////////////////////////						
Net_AO_KC_SHKS04M.top:= haveAlarms();//Нет АО от ШКС					
/////////////////////////////////////////
EGPA_Stop.top:=	(algmanager.mode = modegpa.MODE_STOP); //Режим ЭГПА остановлен							
/////////////////////////////////////////
Avt_SHU_vkl.top:= im.Avtomat_SHU_on.Q;
/////////////////////////////////////////	
All_IM_Off.top:=		(im.mv.onStatus=statusDualInput.STATUS_OFF) 		AND (im.PNS.onStatus=statusDualInput.STATUS_OFF) 			AND (im.nu.nu1.onStatus=statusDualInput.STATUS_OFF) 	AND 
						(im.nu.nu2.onStatus=statusDualInput.STATUS_OFF)		AND (im.v1_Avom.onStatus=statusDualInput.STATUS_OFF) 		AND (im.v2_Avom.onStatus=statusDualInput.STATUS_OFF) 	AND
						(im.v3_Avom.onStatus=statusDualInput.STATUS_OFF) 	AND (im.v4_Avom.onStatus=statusDualInput.STATUS_OFF) 		AND (im.CMN.onStatus=statusDualInput.STATUS_OFF)		AND
						(im.TEN_MB.onStatus=statusDualInput.STATUS_OFF)		AND	(im.TEN_Kollectira.onStatus=statusDualInput.STATUS_OFF)	AND (im.KaloriferAVOM.onStatus=statusDualInput.STATUS_OFF); 
/////////////////////////////////////////							
Nalichie220_SHU_Ai.top:=	(ai.Kontrol_per220V.interval = statusAi.NORMAL)	 AND (ai.Kontrol_post220V.interval = statusAi.NORMAL);				
/////////////////////////////////////////	
BP_Norm.top:= 
		(im.NalichieBP1.Q AND
		im.NalichieBP2.Q AND	
		im.NalichieBP3.Q AND
		im.NalichieBP4.Q AND
		im.NalichieBP5.Q AND
		im.NalichieBP6.Q AND
		im.NalichieBP7_BP8.Q AND
		im.NalichieBP9_BP10.Q AND
		
		im.Nalichie220BEAO.Q AND
		im.NalichiePer220naVhode.Q AND
		im.NalichiePost220naVhode.Q AND
		im.NalichieBP11.Q AND
		im.NalichieBP12.Q);
/////////////////////////////////////////
Naprajenie_U_IM.top:=	im.NalichieU_CMN.q AND im.NalichieU_NU1.Q (*AND im.Nalichie_CU_MV.Q*)  AND im.NalichieU_NU2.Q AND 
						im.NalichieU_PNS.Q; //есть напряжение в цепях управления ИМ
/////////////////////////////////////////
MV_Poloj_RolledON.top:= im.mv.basketStatus = basketStats.BASKET_ROLLEDIN; //Тележка МВ вкачена
/////////////////////////////////////////
MV_Poloj_RolledOFF.top:= im.mv.basketStatus = basketStats.BASKET_ROLLEDOUT; //Тележка МВ выкачена
/////////////////////////////////////////
NOTAnalogNS.top:= NOT (analogsNS()) AND NOT (remont ()); //Нет аналогов неисправных
/////////////////////////////////////////
Net_ASPS_Analogs.top:= (AS_PS_Anologs ()); //Нет АС ПС по Аналогам
/////////////////////////////////////////			
Not_AS.top:=	NOT (protectmanager.anyProtectionSignaling ()); //Нет сработанных защит
/////////////////////////////////////////
Gotov_Vozb.top:= im.VozbutetelisReady.Q;     
/////////////////////////////////////////
Reactornyi_P.top:=im.Reactorni_Pusk.Q AND NOT im.Chastotniy_Pusk.Q;
/////////////////////////////////////////
Chastotnyi_P.top:=im.Chastotniy_Pusk.Q AND NOT im.Reactorni_Pusk.Q;
/////////////////////////////////////////
dP_kr1.top:= ((NOT (im.PerepadDavlenieKran1_Less100.Q)) AND (im.PerepadDavlenieKran1_CK.status = 1));
/////////////////////////////////////////
Auto_Rej.top:=			im.NU1_Automat.Q AND im.PNS_Automat.Q AND im.NU2_Automat.Q;
/////////////////////////////////////////
CK_IM_Norm.top:=	CK_Di();
/////////////////////////////////////////
HAnd_Mode.top:= ((NOT (im.Hand_Reg_rej.Q)) AND (im.Hand_Reg_rej_CK.status = 1));
/////////////////////////////////////////
Impuls_Gaz.top:=(ai.DavlenieImpulsGaz.interval=statusAi.normal);
/////////////////////////////////////////	

	IF		BMP_Err.top AND
			Level_masla_Norm.top AND
			T_masla_Norm.top AND
			Krans_ready_to_move.top AND
			Krans_Poloj.top AND
			Net_AO_KC_SHKS04M.top AND
			EGPA_Stop.top AND
			Avt_SHU_vkl.top AND
			All_IM_Off.top AND
			Nalichie220_SHU_Ai.top AND
			BP_Norm.top AND
			Naprajenie_U_IM.top AND
			MV_Poloj_RolledON.top AND
			NOT MV_Poloj_RolledOFF.top AND
			NOTAnalogNS.top AND 
			Net_ASPS_Analogs.top AND
			Not_AS.top AND
			Gotov_Vozb.top AND
			Chastotnyi_P.top AND
			dP_kr1.top AND
			Auto_Rej.top AND
			CK_IM_Norm.top AND
			HAnd_Mode.top AND
			Impuls_Gaz.top THEN
			ppuFirst_for_Pusk_Ch:= TRUE; ELSE ppuFirst_for_Pusk_Ch:= FALSE; END_IF  //ППУ для первого этапа частотного пуска
			
			
	

IF			BMP_Err.top AND
			Level_masla_Norm.top AND
			T_masla_Norm.top AND
			Krans_ready_to_move.top AND
			Krans_Poloj.top AND
			Net_AO_KC_SHKS04M.top AND
			EGPA_Stop.top AND
			Avt_SHU_vkl.top AND
			All_IM_Off.top AND
			Nalichie220_SHU_Ai.top AND
			BP_Norm.top AND
			Naprajenie_U_IM.top AND
			MV_Poloj_RolledON.top AND
			NOT MV_Poloj_RolledOFF.top AND
			NOTAnalogNS.top AND 
			Net_ASPS_Analogs.top AND
			Not_AS.top AND
			Gotov_Vozb.top AND
			Reactornyi_P.top AND
			dP_kr1.top AND
			Auto_Rej.top AND
			CK_IM_Norm.top AND
			HAnd_Mode.top AND
			Impuls_Gaz.top THEN
			ppuFirst_for_Pusk_R:=TRUE; ELSE ppuFirst_for_Pusk_R:=FALSE; END_IF //первого этапа реакторного пуска
			

	IF		BMP_Err.top AND
			Level_masla_Norm.top AND
			T_masla_Norm.top AND
			Net_AO_KC_SHKS04M.top AND
			EGPA_Stop.top AND
			Avt_SHU_vkl.top AND
			All_IM_Off.top AND
			Nalichie220_SHU_Ai.top AND
			BP_Norm.top AND
			Naprajenie_U_IM.top AND
			MV_Poloj_RolledOFF.top AND
			NOT MV_Poloj_RolledON.top AND
			NOTAnalogNS.top AND 
			Net_ASPS_Analogs.top AND
			Not_AS.top AND
			Auto_Rej.top AND
			CK_IM_Norm.top THEN
			ppuFirst_for_Pms_dPmg:= TRUE; ELSE ppuFirst_for_Pms_dPmg:= FALSE; END_IF//ППУ для проверки масла смазки и масло газ
			

IF			BMP_Err.top AND
			Level_masla_Norm.top AND
			T_masla_Norm.top AND
			Krans_ready_to_move.top AND
			Krans_Poloj.top AND
			Net_AO_KC_SHKS04M.top AND
			EGPA_Stop.top AND
			Avt_SHU_vkl.top AND
			All_IM_Off.top AND
			Nalichie220_SHU_Ai.top AND
			BP_Norm.top AND
			Naprajenie_U_IM.top AND
			MV_Poloj_RolledOFF.top AND
			NOT MV_Poloj_RolledON.top AND
			NOTAnalogNS.top AND 
			Net_ASPS_Analogs.top AND
			Not_AS.top AND
			dP_kr1.top AND
			Auto_Rej.top AND
			CK_IM_Norm.top AND
			Impuls_Gaz.top THEN
			ppuFirst_for_K:=TRUE; ELSE ppuFirst_for_K:=FALSE; END_IF //ППУ проверки кранов
			

IF			BMP_Err.top AND
			Level_masla_Norm.top AND
			T_masla_Norm.top AND
			Krans_ready_to_move.top AND
			Krans_Poloj.top AND
			Net_AO_KC_SHKS04M.top AND
			EGPA_Stop.top AND
			Avt_SHU_vkl.top AND
			All_IM_Off.top AND
			Nalichie220_SHU_Ai.top AND
			BP_Norm.top AND
			Naprajenie_U_IM.top AND
			MV_Poloj_RolledOFF.top AND
			NOT MV_Poloj_RolledON.top AND
			NOTAnalogNS.top AND 
			Net_ASPS_Analogs.top AND
			Not_AS.top AND
			Gotov_Vozb.top AND
			Reactornyi_P.top AND
			dP_kr1.top AND
			Auto_Rej.top AND
			CK_IM_Norm.top AND
			HAnd_Mode.top AND
			Impuls_Gaz.top THEN
			ppuFirst_for_I:=TRUE; ELSE ppuFirst_for_I:=FALSE; END_IF//ППУ имитация пуска


IF			BMP_Err.top AND
			Level_masla_Norm.top AND
			T_masla_Norm.top AND
			Net_AO_KC_SHKS04M.top AND
			EGPA_Stop.top AND
			Avt_SHU_vkl.top AND
			All_IM_Off.top AND
			Nalichie220_SHU_Ai.top AND
			BP_Norm.top AND
			Naprajenie_U_IM.top AND
			MV_Poloj_RolledON.top AND
			NOT MV_Poloj_RolledOFF.top AND
			NOTAnalogNS.top AND 
			Net_ASPS_Analogs.top AND
			Not_AS.top AND
			Gotov_Vozb.top AND
			Chastotnyi_P.top AND
			Auto_Rej.top AND
			CK_IM_Norm.top AND
			HAnd_Mode.top THEN
			ppuFirst_for_V_Ch:=TRUE; ELSE ppuFirst_for_V_Ch:=FALSE;  END_IF


IF			BMP_Err.top AND
			Level_masla_Norm.top AND
			T_masla_Norm.top AND
			Net_AO_KC_SHKS04M.top AND
			EGPA_Stop.top AND
			Avt_SHU_vkl.top AND
			All_IM_Off.top AND
			Nalichie220_SHU_Ai.top AND
			BP_Norm.top AND
			Naprajenie_U_IM.top AND
			MV_Poloj_RolledON.top AND
			NOT MV_Poloj_RolledOFF.top AND
			NOTAnalogNS.top AND 
			Net_ASPS_Analogs.top AND
			Not_AS.top AND
			Gotov_Vozb.top AND
			Reactornyi_P.top AND
			Auto_Rej.top AND
			CK_IM_Norm.top AND
			HAnd_Mode.top THEN
			ppuFirst_for_V_R:=TRUE; ELSE ppuFirst_for_V_R:=FALSE; END_IF
				

	IF		BMP_Err.top AND
			Level_masla_Norm.top AND
			T_masla_Norm.top AND
			Net_AO_KC_SHKS04M.top AND
			Avt_SHU_vkl.top AND
			Nalichie220_SHU_Ai.top AND
			BP_Norm.top AND
			Naprajenie_U_IM.top AND
			MV_Poloj_RolledON.top AND
			NOT MV_Poloj_RolledOFF.top AND
			NOTAnalogNS.top AND 
			Not_AS.top AND
			Gotov_Vozb.top AND
			Chastotnyi_P.top AND
			Auto_Rej.top AND
			HAnd_Mode.top AND ((algmanager.mode=modegpa.MODE_PUSKAP_Ch) OR (algmanager.mode=modegpa.MODE_PUSKPP_Ch) OR (algmanager.mode=modegpa.MODE_PUSKV_Ch)) THEN
			ppuSecond_V_Pusk_Ch:=	TRUE; ELSE ppuSecond_V_Pusk_Ch:= FALSE; END_IF


	IF		BMP_Err.top AND
			Level_masla_Norm.top AND
			T_masla_Norm.top AND
			Net_AO_KC_SHKS04M.top AND
			Avt_SHU_vkl.top AND
			Nalichie220_SHU_Ai.top AND
			BP_Norm.top AND
			Naprajenie_U_IM.top AND
			MV_Poloj_RolledON.top AND
			NOT MV_Poloj_RolledOFF.top AND
			NOTAnalogNS.top AND 
			Not_AS.top AND
			Gotov_Vozb.top AND
			Reactornyi_P.top AND
			Auto_Rej.top AND
			HAnd_Mode.top AND ((algmanager.mode=modegpa.MODE_PUSKAP_R) OR (algmanager.mode=modegpa.MODE_PUSKPP_R) OR (algmanager.mode=modegpa.MODE_PUSKV_R)) THEN
			ppuSecond_V_Pusk_R:=TRUE; ELSE ppuSecond_V_Pusk_R:=	FALSE; END_IF


	IF		BMP_Err.top AND
			Level_masla_Norm.top AND
			T_masla_Norm.top AND
			Net_AO_KC_SHKS04M.top AND
			Avt_SHU_vkl.top AND
			Nalichie220_SHU_Ai.top AND
			BP_Norm.top AND
			Naprajenie_U_IM.top AND
			MV_Poloj_RolledOFF.top AND
			NOT MV_Poloj_RolledON.top AND
			NOTAnalogNS.top AND 
			Not_AS.top AND
			Gotov_Vozb.top AND
			Reactornyi_P.top AND
			Auto_Rej.top AND
			HAnd_Mode.top AND (algmanager.mode=modegpa.MODE_I) THEN
			ppuSecond_I:=	TRUE; ELSE ppuSecond_I:= FALSE; END_IF	//ППУ для второго этапа пуска в режиме "имитация пуска"
			

IF			BMP_Err.top AND
			Level_masla_Norm.top AND
			T_masla_Norm.top AND
			Krans_ready_to_move.top AND
			Krans_Poloj.top AND
			Net_AO_KC_SHKS04M.top AND
			Avt_SHU_vkl.top AND
			Nalichie220_SHU_Ai.top AND
			BP_Norm.top AND
			Naprajenie_U_IM.top AND
			//NOTAnalogNS.top AND 
			Not_AS.top AND
			dP_kr1.top AND
			Auto_Rej.top AND
			Impuls_Gaz.top AND ((algmanager.mode=modegpa.MODE_PUSKAP_R) OR (algmanager.mode=modegpa.MODE_PUSKPP_R) OR 
								(algmanager.mode=modegpa.MODE_PUSKAP_Ch) OR (algmanager.mode=modegpa.MODE_PUSKPP_Ch) OR
								(algmanager.mode=modegpa.MODE_I) OR (algmanager.mode=modegpa.MODE_PUSKK)) THEN
								ppuThird:=TRUE; ELSE ppuThird:=FALSE;	END_IF//ППУ для третьего этапа пуска
			

	IF		(NOT (im.kran6.so OR im.kran6.sz OR
			im.kran4.so OR im.kran4.sz)) AND
			(Im.kran6.onStatus=statusDualInput.STATUS_ON) AND 
			(Im.kran4.onStatus=statusDualInput.STATUS_ON) AND 
			Net_AO_KC_SHKS04M.top AND (NOT remont ()) AND
			(Im.kran1.onStatus=statusDualInput.STATUS_On) AND
			(Im.kran2.onStatus=statusDualInput.STATUS_On) AND
			Impuls_Gaz.top AND ((algmanager.mode=modegpa.MODE_PUSKAP_R) OR (algmanager.mode=modegpa.MODE_PUSKPP_R) OR 
								(algmanager.mode=modegpa.MODE_PUSKAP_Ch) OR (algmanager.mode=modegpa.MODE_PUSKPP_Ch) OR
								(algmanager.mode=modegpa.MODE_I) OR (algmanager.mode=modegpa.MODE_PUSKK)) THEN
								ppuForth:=TRUE; ELSE ppuForth:=FALSE; END_IF	//ППУ для четвертого этапа пуска

METHOD PRIVATE AS_PS_Anologs : BOOL
VAR_INPUT
END_VAR

 AS_PS_Anologs:= 	(ai.TMediStatoraKanall.interval 								= statusAi.NORMAL) 	AND 
 				 	(ai.TMediStatoraKanal2.interval 								= statusAi.NORMAL) 	AND
				 	(ai.TMediStatoraKanal3.interval 								= statusAi.NORMAL) 	AND
				 	(ai.TStalisStatoraKanall.interval 								= statusAi.NORMAL) 	AND
				 	(ai.TStalisStatoraKanal2.interval 								= statusAi.NORMAL) 	AND
				 	(ai.TStalisStatoraKanal3.interval 								= statusAi.NORMAL) 	AND
				 	(ai.TGorjachegoVozduhaEDKanall.interval 						= statusAi.NORMAL) 	AND
				 	(ai.TGorjachegoVozduhaEDKanal2.interval 						= statusAi.NORMAL) 	AND
				 	(ai.THolodnogoVozduhaEDKanall.interval 							= statusAi.NORMAL) 	AND
				 	(ai.THolodnogoVozduhaEDKanal2.interval 							= statusAi.NORMAL) 	AND
				 	(ai.TOpornogoPodshipnikaEDT_1.interval 							= statusAi.NORMAL) 	AND
					(ai.TOpornoYpornogoPodshipnikaEDT_2.interval 					= statusAi.NORMAL) 	AND
					(ai.TOpornoYpornogoPodshipnikaKolesaRedEDT_3.interval 			= statusAi.NORMAL) 	AND
					(ai.TOpornoYpornogoPodshipnikaKolesaRedHT_4.interval 			= statusAi.NORMAL) 	AND
					(ai.TOpornogoPodshipnikaShesterniReduktoraT_5.interval 			= statusAi.NORMAL) 	AND
					(ai.TOpornogoPodshipnikaReduktoraHT_6.interval 					= statusAi.NORMAL) 	AND
					(ai.TOpornoYpornogoPodshipnikaNagnetateljaT_7_1.interval 		= statusAi.NORMAL) 	AND
					(ai.TOpornoYpornogoPodshipnikaNagnetateljaT_7_2.interval 		= statusAi.NORMAL) 	AND
					(ai.TOpornoYpornogoPodshipnikaSvobodnogoKoncaNT_8_1.interval 	= statusAi.NORMAL) 	AND
					(ai.TOpornoYpornogoPodshipnikaSvobodnogoKoncaNT_8_2.interval 	= statusAi.NORMAL) 	AND
					(ai.TYpornogoPodshipnikaRavKolodokHT_9_1.interval 				= statusAi.NORMAL) 	AND
					(ai.TYpornogoPodshipnikaRavKolodokHT_9_2.interval 				= statusAi.NORMAL) 	AND
					(ai.TYpornogoPodshipnikaNerabKolodokHT_10_1.interval 			= statusAi.NORMAL) 	AND
					(ai.TYpornogoPodshipnikaNerabKolodokHT_10_2.interval 			= statusAi.NORMAL) 	AND
					(ai.TgazaNaVhodeH.interval 										= statusAi.NORMAL) 	AND
					(ai.TgazaNaVyhodeH.interval 									= statusAi.NORMAL) 	AND
					(ai.TMasladoAVOM.interval 										= statusAi.NORMAL) 	AND
					(ai.TMaslaPosleAVOM.interval 									= statusAi.NORMAL) 	AND
					(ai.TMaslaMB.interval 											= statusAi.NORMAL) 	AND
					(ai.TMaslaMB_TEN.interval 										= statusAi.NORMAL) 	AND			
					(ai.VibroSkorostOPED_T1.interval 								= statusAi.NORMAL) 	AND
					(ai.VibroSkorostOYPED_T2.interval 								= statusAi.NORMAL) 	AND
					(ai.VibroSkorostOYPKolesaED_T3.interval 						= statusAi.NORMAL) 	AND
					(ai.VibroSkorostOPKolesaRH_T4.interval 							= statusAi.NORMAL) 	AND
					(ai.VibroSkorostOPShesterniRED_T5.interval 						= statusAi.NORMAL) 	AND
					(ai.VibroSkorostOPShesterniReduktoraH_T6.interval 				= statusAi.NORMAL) 	AND
					(ai.OsSdvigNagnetatelja_Plus.interval 							= statusAi.NORMAL) 	AND
					(ai.OsSdvigNagnetatelja_Minus.interval 							= statusAi.NORMAL);
END_METHOD

METHOD PRIVATE haveAlarms : BOOL
VAR_INPUT
	
END_VAR

haveAlarms:= (NOT (Im.AOKC_SHKC.Q)) AND (im.AOKC_SHKC_CK.status = 1);
END_METHOD

METHOD PUBLIC reset
VAR_INPUT
END_VAR
SUPER^.reset();
ppuFirst_for_Pusk_Ch:=FALSE;
ppuFirst_for_Pusk_R:=FALSE;
ppuFirst_for_V_Ch:=FALSE;
ppuFirst_for_V_R:=FALSE;
ppuFirst_for_Pms_dPmg:=FALSE;
ppuFirst_for_K:=FALSE;
ppuFirst_for_I:=FALSE;
ppuSecond_V_Pusk_Ch:=FALSE;
ppuSecond_V_Pusk_R:=FALSE;
ppuSecond_I:=FALSE;
ppuThird:=FALSE;
ppuForth:=FALSE;
statusSet.setBit(15,FALSE); //к пуску готов
statusSet.setBit(16, FALSE); //к проверкам готов
statusSet.setBit(17,FALSE); //ко 2-му этапу пуска готов
statusSet.setBit(18,FALSE); //ко 3-му этапу пуска готов
statusSet.setBit(19,FALSE); //к 4-му этапу пуска готов
statusSet.setBit(20,FALSE); //к 4-му этапу пуска готов
END_METHOD

METHOD PUBLIC writeImStatus
VAR_INPUT
END_VAR
SUPER^.writeImStatus();

statusSet.setBit(15,ppuFirst_for_Pusk_Ch); //к пуску частотному
statusSet.setBit(16,ppuFirst_for_Pusk_r); //к пуску реакторному
statusSet.setBit(17,(ppuFirst_for_V_Ch OR ppuFirst_for_V_r OR ppuFirst_for_Pms_dPmg OR ppuFirst_for_K OR ppuFirst_for_I)); //к проверкам готов
statusSet.setBit(18,(ppuSecond_V_Pusk_ch OR ppuSecond_V_Pusk_r OR ppuSecond_I)); //ко 2-му этапу пуска готов
statusSet.setBit(19,(ppuThird)); //к 3-му этапу пуска готов
statusSet.setBit(20,(ppuForth)); //к 4-му этапу пуска готов
END_METHOD

METHOD PUBLIC Remont : BOOL
VAR_INPUT
END_VAR
Remont := protections.p_TOpornogoPodshipnikaEDT_1.remont OR

	
		
		protections.p_TOpornoYpornogoPodshipnikaEDT_2.remont OR
		protections.p_TOpornoYpornogoPodshipnikaKolesaRedEDT_3.remont OR
		protections.p_TOpornoYpornogoPodshipnikaKolesaRedHT_4.remont OR
		protections.p_TOpornogoPodshipnikaShesterniReduktoraT_5.remont OR
		protections.p_TOpornogoPodshipnikaReduktoraHT_6.remont OR
		protections.p_TOpornoYpornogoPodshipnikaNagnetateljaT_7.remont OR
		protections.p_TOpornoYpornogoPodshipnikaSvobodnogoKoncaNT_8.remont OR
		protections.p_TYpornogoPodshipnikaRavKolodokHT_9.remont OR
		protections.p_TYpornogoPodshipnikaNerabKolodokHT_10.remont OR
		protections.p_TgazaNaVyhodeH.remont OR
		
	(*Давления*)
		
		protections.p_OsSdvigNagnetatelja_Plus.remont OR
		protections.p_OsSdvigNagnetatelja_Minus.remont OR
		protections.p_DGazaNaVhodeNagnetatelja_GPA_STOP.remont OR
		protections.p_DGazaNaVyhodeNagnetatelja_GPA_STOP.remont OR
		//protections.p_DGazaNaVhodeNagnetatelja.remont OR
		protections.p_DGazaNaVyhodeNagnetatelja.remont OR
		protections.p_PerepadDavlenieMasloGaz.remont OR
		protections.p_DavlenijaMasloSmNizkoe.remont OR
		protections.p_DavlenijaMasloSmVysokoe.remont OR
	
	(*Вибрация*)
		
		protections.p_VibroSkorostOPED_T1.remont OR
		protections.p_VibroSkorostOYPED_T2.remont OR
		protections.p_VibroSkorostOYPKolesaED_T3.remont OR
		protections.p_VibroSkorostOPKolesaRH_T4.remont OR
		protections.p_VibroSkorostOPShesterniRED_T5.remont OR
		protections.p_VibroSkorostOPShesterniReduktoraH_T6.remont OR
	(*Дискретные сигналы *)
		
		protections.p_PerepadDavlenieMasloGaz_Less100.remont OR
		protections.p_RegVozbOff.remont OR
		protections.p_Fail_Chastotniy_Pusk.remont OR
		protections.p_OFFAvarSwitch.remont OR
		protections.p_AOKC_SHKC.remont OR
		protections.p_AO_PRU.remont OR
		protections.p_AO_fromSHU.remont OR	
					
(*Защиты по ИМ *)																							
		protections.p_mvOff.remont OR
		protections.p_kran1.remont OR
		protections.p_kran2.remont;
END_METHOD

METHOD PUBLIC analogsNs : BOOL
VAR_INPUT
END_VAR
VAR
		
END_VAR
SUPER^();
analogsNs:=
	
		(ai.TStalisStatoraKanall.interval 											< statusAi.NORMAL) 	OR
		(ai.TStalisStatoraKanal2.interval 											< statusAi.NORMAL) 	OR
		(ai.TStalisStatoraKanal3.interval 											< statusAi.NORMAL) 	OR
		(ai.TMediStatoraKanall.interval 											< statusAi.NORMAL) 	OR
		(ai.TMediStatoraKanal2.interval 											< statusAi.NORMAL) 	OR
		(ai.TMediStatoraKanal3.interval 											< statusAi.NORMAL) 	OR
		(ai.TOpornogoPodshipnikaEDT_1.interval 										< statusAi.NORMAL) 	OR
		(ai.TOpornoYpornogoPodshipnikaEDT_2.interval 								< statusAi.NORMAL) 	OR
		(ai.TOpornoYpornogoPodshipnikaKolesaRedEDT_3.interval 						< statusAi.NORMAL) 	OR
		(ai.TOpornoYpornogoPodshipnikaKolesaRedHT_4.interval 						< statusAi.NORMAL) 	OR
		(ai.TOpornogoPodshipnikaShesterniReduktoraT_5.interval 						< statusAi.NORMAL) 	OR
		(ai.TOpornogoPodshipnikaReduktoraHT_6.interval 								< statusAi.NORMAL) 	OR
		(ai.TOpornoYpornogoPodshipnikaNagnetateljaT_7_1.interval 					< statusAi.NORMAL) 	OR
		(ai.TOpornoYpornogoPodshipnikaNagnetateljaT_7_2.interval 					< statusAi.NORMAL) 	OR
		(ai.TOpornoYpornogoPodshipnikaSvobodnogoKoncaNT_8_1.interval 				< statusAi.NORMAL) 	OR
		(ai.TOpornoYpornogoPodshipnikaSvobodnogoKoncaNT_8_2.interval 				< statusAi.NORMAL) 	OR
		(ai.TYpornogoPodshipnikaRavKolodokHT_9_1.interval 							< statusAi.NORMAL) 	OR
		(ai.TYpornogoPodshipnikaRavKolodokHT_9_2.interval 							< statusAi.NORMAL) 	OR
		(ai.TYpornogoPodshipnikaNerabKolodokHT_10_1.interval 						< statusAi.NORMAL) 	OR
		(ai.TYpornogoPodshipnikaNerabKolodokHT_10_2.interval 						< statusAi.NORMAL) 	OR
		(ai.THolodnogoVozduhaEDKanall.interval 										< statusAi.NORMAL) 	OR
		(ai.THolodnogoVozduhaEDKanal2.interval 										< statusAi.NORMAL) 	OR
		(ai.TGorjachegoVozduhaEDKanall.interval 									< statusAi.NORMAL) 	OR
		(ai.TGorjachegoVozduhaEDKanal2.interval 									< statusAi.NORMAL) 	OR
		(ai.TgazaNaVhodeH.interval 													< statusAi.NORMAL) 	OR
		(ai.TgazaNaVyhodeH.interval 												< statusAi.NORMAL) 	OR
		(ai.TMasladoAVOM.interval 													< statusAi.NORMAL) 	OR
		(ai.TMaslaPosleAVOM.interval 												< statusAi.NORMAL) 	OR
		(ai.TMaslaMB.interval 														< statusAi.NORMAL) 	OR
		(ai.TMaslaMB_TEN.interval 													< statusAi.NORMAL) 	OR
		(ai.DavlenijaMasloSmNizkoe.interval 										< statusAi.NORMAL) 	OR
		(ai.PerepadDavlenieNaMasloFiltre.interval 									< statusAi.NORMAL) 	OR
		(ai.DavlenijaMasloSmVysokoe.interval 										< statusAi.NORMAL) 	OR
		(ai.DavlenijaMaslaPosleGNS.interval 										< statusAi.NORMAL) 	OR
		(ai.DavlenijaMaslaPosleNU.interval 											< statusAi.NORMAL) 	OR
		(ai.PerepadDavlenieNaKonfuzore.interval 									< statusAi.NORMAL) 	OR
		(ai.OsSdvigNagnetatelja_Plus.interval 										< statusAi.NORMAL) 	OR
		(ai.OsSdvigNagnetatelja_Minus.interval 										< statusAi.NORMAL) 	OR
		(ai.PerepadDavlenieMasloGaz.interval 										< statusAi.NORMAL) 	OR
		(ai.DGazaNaVhodeNagnetatelja.interval 										< statusAi.NORMAL) 	OR
		(ai.DGazaNaVyhodeNagnetatelja.interval 										< statusAi.NORMAL) 	OR
		(ai.DavlenieImpulsGaz.interval 												< statusAi.NORMAL) 	OR
		(ai.YrovenMaslaMB.interval 													< statusAi.NORMAL) 	OR
		(ai.Kontrol_per220V.interval 												< statusAi.NORMAL) 	OR
		(ai.Kontrol_post220V.interval 												< statusAi.NORMAL) 	OR
		(ai.VibroSkorostOPED_T1.interval 											< statusAi.NORMAL) 	OR
		(ai.VibroSkorostOYPED_T2.interval 											< statusAi.NORMAL) 	OR
		(ai.VibroSkorostOYPKolesaED_T3.interval 									< statusAi.NORMAL) 	OR
		(ai.VibroSkorostOPKolesaRH_T4.interval 										< statusAi.NORMAL) 	OR
		(ai.VibroSkorostOPShesterniRED_T5.interval 									< statusAi.NORMAL) 	OR
		(ai.VibroSkorostOPShesterniReduktoraH_T6.interval 							< statusAi.NORMAL) 	OR
		(ai.TokStatora.interval 													< statusAi.NORMAL) ;
END_METHOD

METHOD PUBLIC CK_Di : BOOL
VAR_INPUT
END_VAR

 CK_Di:=	(im.PerepadDavlenieMasloGaz_CK.status = 1)	AND
 			(im.PerepadDavlenieKran1_CK.status = 1)		AND
			(im.LevelMaslaAkkum_CK.status = 1)			AND
			(im.LoadDriveisGranted_CK.status = 1)		AND
			(im.VozbutetelisReady_CK.status = 1)			AND
			(im.RegVozbOff_CK.status = 1)				AND
			(im.MainRegOff_CK.status = 1)				AND
			(im.AVR_Vozb_Malfanctional_CK.status = 1)		AND
			(im.OFFAvarSwitch_CK.status = 1)				AND
			(im.AsynchronnyHod_CK.status = 1)		AND
			(im.Avtomat_SHU_on_CK.status = 1)		AND
			(im.Avtomat_SHP_on_CK.status = 1)			AND
			(im.U_Sekcii_CK.status = 1)					AND
			(im.Reactorni_Pusk_CK.status = 1)				AND
			(im.Chastotniy_Pusk_CK.status = 1)			AND
			(im.Fail_Chastotniy_Pusk_CK.status = 1)		AND
			(im.Hand_Reg_rej_CK.status = 1)				AND
			(im.AOKC_SHKC_CK.status = 1)					AND
			(im.NO_fromSHU_CK.status = 1)					AND
			(im.AO_fromSHU_CK.status = 1)					AND
			(im.AO_PRU_CK.status = 1)						AND
			(im.NKU_1_On_CK.status = 1)					AND
			(im.NKU_2_On_CK.status = 1)					AND
			(im.MVvkl_NAlichie_CK.status = 1)				AND
			(im.MVvykl_NAlichie_CK.status = 1)			AND
			(im.MVControl_Work_NAlichie_CK.status = 1)		AND
			(im.PNS_vkl_NAlichie_CK.status = 1)			AND
			(im.NU1_vkl_NAlichie_CK.status = 1)			AND
			(im.NU2_vkl_NAlichie_CK.status = 1)			AND
			(im.AVOM1_vkl_NAlichie_CK.status = 1)			AND
			(im.AVOM2_vkl_NAlichie_CK.status = 1)			AND
			(im.AVOM3_vkl_NAlichie_CK.status = 1)			AND
			(im.AVOM4_vkl_NAlichie_CK.status = 1)			AND
			(im.TEN_MB_vkl_NAlichie_CK.status = 1)			AND
			(im.TEN_Kollectora_vkl_NAlichie_CK.status = 1)	AND
			(im.Kalorifer_AVOM_vkl_NAlichie_CK.status = 1)	AND
			(im.CMN_vkl_NAlichie_CK.status = 1) AND (im.kran1.onstatus<>statusDualInput.STATUS_ERROR)
			AND (im.kran2.onstatus<>statusDualInput.STATUS_ERROR) AND (im.kran3.onstatus<>statusDualInput.STATUS_ERROR)
			AND (im.kran3b.onstatus<>statusDualInput.STATUS_ERROR) AND (im.kran4.onstatus<>statusDualInput.STATUS_ERROR)
			AND (im.kran5.onstatus<>statusDualInput.STATUS_ERROR)	AND (im.kran6.onstatus<>statusDualInput.STATUS_ERROR);
END_METHOD

METHOD PUBLIC Neisp_DI : BOOL
VAR_INPUT
END_VAR
Neisp_DI:= 
		((ystavki.dPmg_Rassogl.status = 1) OR
		im.NalichieBP1_NS.Q OR
		im.NalichieBP2_NS.Q OR
		im.NalichieBP3_NS.Q OR
		im.NalichieBP4_NS.Q OR
		im.NalichieBP5_NS.Q OR
		im.NalichieBP6_NS.Q OR
		im.NalichieBP7_BP8_NS.Q OR
		im.NalichieBP9_BP10_NS.Q OR
		im.Nalichie_CU_MV_NS.Q OR
		im.Nalichie220BEAO_NS.Q OR
		im.NalichiePer220naVhode_NS.Q OR
		im.NalichiePost220naVhode_NS.Q OR
		im.NalichieBP11_NS.Q OR
		im.NalichieBP12_NS.Q OR
		im.NET_U_PNS.Q OR
		im.NET_U_CMN.Q OR
		im.NET_U_NU1.Q OR
		im.NET_U_NU2.Q OR
 		im.kran1.sdvig OR
		im.kran2.sdvig OR
		im.kran3.sdvig OR
		im.kran3b.sdvig OR
		im.kran4.sdvig OR
		im.kran5.sdvig OR
		im.kran6.sdvig OR
		(im.LevelMaslaAkkum.status = 1) OR
		im.MainRegOff.Q OR
		im.AVR_Vozb_Malfanctional.Q OR
		im.AsynchronnyHod.Q);
END_METHOD

END_FUNCTION_BLOCK

// K2/std12k5/Pusk/ppuAlg
	{attribute 'symbol' := 'none'}
FUNCTION_BLOCK ppuAlg EXTENDS StepBySteapAlgoritm
VAR_INPUT
END_VAR
VAR_OUTPUT
	{attribute 'symbol' := 'read'}
	ppuFirst_for_Pusk_Ch:BOOL;
	{attribute 'symbol' := 'read'}
	ppuFirst_for_Pusk_R:BOOL;
	{attribute 'symbol' := 'read'}
	ppuFirst_for_V_Ch:BOOL;
	{attribute 'symbol' := 'read'}
	ppuFirst_for_V_R:BOOL;
	{attribute 'symbol' := 'read'}
	ppuFirst_for_Pms_dPmg: BOOL;
	{attribute 'symbol' := 'read'}
	ppuFirst_for_K: BOOL;
	{attribute 'symbol' := 'read'}
	ppuFirst_for_I: BOOL;
	{attribute 'symbol' := 'read'}
	ppuSecond_V_Pusk_Ch: BOOL;
	{attribute 'symbol' := 'read'}
	ppuSecond_V_Pusk_R: BOOL;
	{attribute 'symbol' := 'read'}
	ppuSecond_I: BOOL;
	{attribute 'symbol' := 'read'}
	ppuThird:BOOL;
	{attribute 'symbol' := 'read'}
	ppuForth:BOOL;
END_VAR
VAR
	BMP_Err:					CustomPhase (table:=ADR(phasesTable)):=		(phaseNumber:=0); //Все аналоги исправны
	
	Level_masla_Norm: 			CustomPhase (table:=ADR(phasesTable)):=		(phaseNumber:=1); //уровень масла в МЮ нормальный
	
	T_masla_Norm: 				CustomPhase (table:=ADR(phasesTable)):=		(phaseNumber:=2); //температура масла в мб больше 25
	
	Krans_ready_to_move:		CustomPhase (table:=ADR(phasesTable)):=		(phaseNumber:=3); //Краны готовы к управлению
	
	Krans_Poloj:				CustomPhase (table:=ADR(phasesTable)):=		(phaseNumber:=4); //Положение кранов соответствует ППУ
	
	Net_AO_KC_SHKS04M: 			CustomPhase (table:=ADR(phasesTable)):=		(phaseNumber:=5); //Нет АО от ШКС
	
	EGPA_Stop:					CustomPhase (table:=ADR(phasesTable)):=		(phaseNumber:=6); //ЭГПА остановлен
	
	Avt_SHU_vkl:				CustomPhase (table:=ADR(phasesTable)):=		(phaseNumber:=7); //Автомат в ячейке ШУ включен
	
	All_IM_Off:					CustomPhase (table:=ADR(phasesTable)):=		(phaseNumber:=8); //Все ИМ выключены
	
	Nalichie220_SHU_Ai:			CustomPhase (table:=ADR(phasesTable)):=		(phaseNumber:=9); //Напряжение в ШУ в норме по AI
	
	BP_Norm:					CustomPhase (table:=ADR(phasesTable)):=		(phaseNumber:=10); //Все БП исправны
	
	Naprajenie_U_IM: 			CustomPhase (table:=ADR(phasesTable)):=		(phaseNumber:=11); //есть напряжение в цепях управления ИМ
	
	MV_Poloj_RolledON:			CustomPhase (table:=ADR(phasesTable)):=		(phaseNumber:=12); //Тележка МВ вкачена
	
	MV_Poloj_RolledOFF:			CustomPhase (table:=ADR(phasesTable)):=		(phaseNumber:=13); //Тележка МВ выкачена 
	
	NOTAnalogNS: 				CustomPhase (table:=ADR(phasesTable)):=		(phaseNumber:=14); //Все аналоги исправны
	
	Net_ASPS_Analogs:			CustomPhase (table:=ADR(phasesTable)):=		(phaseNumber:=15); //Нет АС и ПС по аналогам
	
	Not_AS:						CustomPhase (table:=ADR(phasesTable)):=		(phaseNumber:=16); //Нет сработанных защит
	
	Gotov_Vozb:					CustomPhase (table:=ADR(phasesTable)):=		(phaseNumber:=17); //Возбудитель Готов
	
	Reactornyi_P:				CustomPhase (table:=ADR(phasesTable)):=		(phaseNumber:=18); //Реакторный пуск
	
	Chastotnyi_P:				CustomPhase (table:=ADR(phasesTable)):=		(phaseNumber:=19); //Частотный пуск
	
	dP_kr1:						CustomPhase (table:=ADR(phasesTable)):=		(phaseNumber:=20); //Перепад на кране один есть
	
	Auto_Rej:					CustomPhase (table:=ADR(phasesTable)):=		(phaseNumber:=21); //ПНС, НУ в автоматическом режиме
	
	CK_IM_Norm: 				CustomPhase (table:=ADR(phasesTable)):=		(phaseNumber:=22); //Цепи контроля ИМ исправны
	
	HAnd_Mode:					CustomPhase (table:=ADR(phasesTable)):=		(phaseNumber:=23); //Ручной режим
	
	Impuls_Gaz:					CustomPhase (table:=ADR(phasesTable)):=		(phaseNumber:=24); //импульсный газ	
	
END_VAR

SUPER^();
BMP_Err.top:= ((BMPERR_k = 0) OR (kontroller.imit));
/////////////////////////////////////////
Level_masla_Norm.top:=(ai.YrovenMaslaMB.interval=statusAi.normal);//уровень масла в норме
/////////////////////////////////////////
T_masla_Norm.top:=(ai.TMaslaMB.interval=statusAi.normal);//температура масла в норме
/////////////////////////////////////////
Krans_ready_to_move.top:= 	NOT (im.kran1.so OR im.kran1.sz OR im.kran2.so OR im.kran2.sz OR im.kran3.so OR im.kran3.sz OR im.kran3b.so OR im.kran3b.sz OR im.kran4.so OR im.kran4.sz OR
							im.kran5.so OR im.kran5.sz OR im.kran6.so OR im.kran6.sz); //Краны готовы к управлению
/////////////////////////////////////////
Krans_Poloj.top:=		(Im.kran1.onStatus=statusDualInput.STATUS_OFF) AND
						(Im.kran2.onStatus=statusDualInput.STATUS_OFF) AND
						(Im.kran3.onStatus=statusDualInput.STATUS_OFF) AND
						(Im.kran3b.onStatus=statusDualInput.STATUS_ON) AND
						(Im.kran4.onStatus=statusDualInput.STATUS_OFF) AND
						(Im.kran5.onStatus=statusDualInput.STATUS_ON) AND 
						(Im.kran6.onStatus=statusDualInput.STATUS_ON); 
/////////////////////////////////////////						
Net_AO_KC_SHKS04M.top:= haveAlarms();//Нет АО от ШКС					
/////////////////////////////////////////
EGPA_Stop.top:=	(algmanager.mode = modegpa.MODE_STOP); //Режим ЭГПА остановлен							
/////////////////////////////////////////
Avt_SHU_vkl.top:= im.Avtomat_SHU_on.Q;
/////////////////////////////////////////	
All_IM_Off.top:=		(im.mv.onStatus=statusDualInput.STATUS_OFF) 		AND (im.PNS.onStatus=statusDualInput.STATUS_OFF) 			AND (im.nu.nu1.onStatus=statusDualInput.STATUS_OFF) 	AND 
						(im.nu.nu2.onStatus=statusDualInput.STATUS_OFF)		AND (im.v1_Avom.onStatus=statusDualInput.STATUS_OFF) 		AND (im.v2_Avom.onStatus=statusDualInput.STATUS_OFF) 	AND
						(im.v3_Avom.onStatus=statusDualInput.STATUS_OFF) 	AND (im.v4_Avom.onStatus=statusDualInput.STATUS_OFF) 		AND (im.CMN.onStatus=statusDualInput.STATUS_OFF)		AND
						(im.TEN_MB.onStatus=statusDualInput.STATUS_OFF)		AND	(im.TEN_Kollectira.onStatus=statusDualInput.STATUS_OFF)	AND (im.KaloriferAVOM.onStatus=statusDualInput.STATUS_OFF); 
/////////////////////////////////////////							
Nalichie220_SHU_Ai.top:=	(ai.Kontrol_per220V.interval = statusAi.NORMAL)	 AND (ai.Kontrol_post220V.interval = statusAi.NORMAL);				
/////////////////////////////////////////	
BP_Norm.top:= 
		(im.NalichieBP1.Q AND
		im.NalichieBP2.Q AND	
		im.NalichieBP3.Q AND
		im.NalichieBP4.Q AND
		im.NalichieBP5.Q AND
		im.NalichieBP6.Q AND
		im.NalichieBP7_BP8.Q AND
		im.NalichieBP9_BP10.Q AND
		
		im.Nalichie220BEAO.Q AND
		im.NalichiePer220naVhode.Q AND
		im.NalichiePost220naVhode.Q AND
		im.NalichieBP11.Q AND
		im.NalichieBP12.Q);
/////////////////////////////////////////
Naprajenie_U_IM.top:=	im.NalichieU_CMN.q (*AND im.Nalichie_CU_MV.Q*) AND im.NalichieU_NU1.Q AND im.NalichieU_NU2.Q AND 
						im.NalichieU_PNS.Q; //есть напряжение в цепях управления ИМ
/////////////////////////////////////////
MV_Poloj_RolledON.top:= im.mv.basketStatus = basketStats.BASKET_ROLLEDIN; //Тележка МВ вкачена
/////////////////////////////////////////
MV_Poloj_RolledOFF.top:= im.mv.basketStatus = basketStats.BASKET_ROLLEDOUT; //Тележка МВ выкачена
/////////////////////////////////////////
NOTAnalogNS.top:= NOT (analogsNS()) AND NOT (remont ()); //Нет аналогов неисправных
/////////////////////////////////////////
Net_ASPS_Analogs.top:= (AS_PS_Anologs ()); //Нет АС ПС по Аналогам
/////////////////////////////////////////			
Not_AS.top:=	NOT (protectmanager.anyProtectionSignaling ()); //Нет сработанных защит
/////////////////////////////////////////
Gotov_Vozb.top:= im.VozbutetelisReady.Q;     
/////////////////////////////////////////
Reactornyi_P.top:=im.Reactorni_Pusk.Q AND NOT im.Chastotniy_Pusk.Q;
/////////////////////////////////////////
Chastotnyi_P.top:=im.Chastotniy_Pusk.Q AND NOT im.Reactorni_Pusk.Q;
/////////////////////////////////////////
dP_kr1.top:= ((NOT (im.PerepadDavlenieKran1_Less100.Q)) AND (im.PerepadDavlenieKran1_CK.status = 1));
/////////////////////////////////////////
Auto_Rej.top:=			im.NU1_Automat.Q AND im.PNS_Automat.Q AND im.NU2_Automat.Q;
/////////////////////////////////////////
CK_IM_Norm.top:=	CK_Di();
/////////////////////////////////////////
HAnd_Mode.top:= ((NOT (im.Hand_Reg_rej.Q)) AND (im.Hand_Reg_rej_CK.status = 1));
/////////////////////////////////////////
Impuls_Gaz.top:=(ai.DavlenieImpulsGaz.interval=statusAi.normal);
/////////////////////////////////////////	

	IF		BMP_Err.top AND
			Level_masla_Norm.top AND
			T_masla_Norm.top AND
			Krans_ready_to_move.top AND
			Krans_Poloj.top AND
			Net_AO_KC_SHKS04M.top AND
			EGPA_Stop.top AND
			Avt_SHU_vkl.top AND
			All_IM_Off.top AND
			Nalichie220_SHU_Ai.top AND
			BP_Norm.top AND
			Naprajenie_U_IM.top AND
			MV_Poloj_RolledON.top AND
			NOT MV_Poloj_RolledOFF.top AND
			NOTAnalogNS.top AND 
			Net_ASPS_Analogs.top AND
			Not_AS.top AND
			Gotov_Vozb.top AND
			Chastotnyi_P.top AND
			dP_kr1.top AND
			Auto_Rej.top AND
			CK_IM_Norm.top AND
			HAnd_Mode.top AND
			Impuls_Gaz.top THEN
			ppuFirst_for_Pusk_Ch:= TRUE; ELSE ppuFirst_for_Pusk_Ch:= FALSE; END_IF  //ППУ для первого этапа частотного пуска
			
			
	

IF			BMP_Err.top AND
			Level_masla_Norm.top AND
			T_masla_Norm.top AND
			Krans_ready_to_move.top AND
			Krans_Poloj.top AND
			Net_AO_KC_SHKS04M.top AND
			EGPA_Stop.top AND
			Avt_SHU_vkl.top AND
			All_IM_Off.top AND
			Nalichie220_SHU_Ai.top AND
			BP_Norm.top AND
			Naprajenie_U_IM.top AND
			MV_Poloj_RolledON.top AND
			NOT MV_Poloj_RolledOFF.top AND
			NOTAnalogNS.top AND 
			Net_ASPS_Analogs.top AND
			Not_AS.top AND
			Gotov_Vozb.top AND
			Reactornyi_P.top AND
			dP_kr1.top AND
			Auto_Rej.top AND
			CK_IM_Norm.top AND
			HAnd_Mode.top AND
			Impuls_Gaz.top THEN
			ppuFirst_for_Pusk_R:=TRUE; ELSE ppuFirst_for_Pusk_R:=FALSE; END_IF //первого этапа реакторного пуска
			

	IF		BMP_Err.top AND
			Level_masla_Norm.top AND
			T_masla_Norm.top AND
			Net_AO_KC_SHKS04M.top AND
			EGPA_Stop.top AND
			Avt_SHU_vkl.top AND
			All_IM_Off.top AND
			Nalichie220_SHU_Ai.top AND
			BP_Norm.top AND
			Naprajenie_U_IM.top AND
			MV_Poloj_RolledOFF.top AND
			NOT MV_Poloj_RolledON.top AND
			NOTAnalogNS.top AND 
			Net_ASPS_Analogs.top AND
			Not_AS.top AND
			Auto_Rej.top AND
			CK_IM_Norm.top THEN
			ppuFirst_for_Pms_dPmg:= TRUE; ELSE ppuFirst_for_Pms_dPmg:= FALSE; END_IF//ППУ для проверки масла смазки и масло газ
			

IF			BMP_Err.top AND
			Level_masla_Norm.top AND
			T_masla_Norm.top AND
			Krans_ready_to_move.top AND
			Krans_Poloj.top AND
			Net_AO_KC_SHKS04M.top AND
			EGPA_Stop.top AND
			Avt_SHU_vkl.top AND
			All_IM_Off.top AND
			Nalichie220_SHU_Ai.top AND
			BP_Norm.top AND
			Naprajenie_U_IM.top AND
			MV_Poloj_RolledOFF.top AND
			NOT MV_Poloj_RolledON.top AND
			NOTAnalogNS.top AND 
			Net_ASPS_Analogs.top AND
			Not_AS.top AND
			dP_kr1.top AND
			Auto_Rej.top AND
			CK_IM_Norm.top AND
			Impuls_Gaz.top THEN
			ppuFirst_for_K:=TRUE; ELSE ppuFirst_for_K:=FALSE; END_IF //ППУ проверки кранов
			

IF			BMP_Err.top AND
			Level_masla_Norm.top AND
			T_masla_Norm.top AND
			Krans_ready_to_move.top AND
			Krans_Poloj.top AND
			Net_AO_KC_SHKS04M.top AND
			EGPA_Stop.top AND
			Avt_SHU_vkl.top AND
			All_IM_Off.top AND
			Nalichie220_SHU_Ai.top AND
			BP_Norm.top AND
			Naprajenie_U_IM.top AND
			MV_Poloj_RolledOFF.top AND
			NOT MV_Poloj_RolledON.top AND
			NOTAnalogNS.top AND 
			Net_ASPS_Analogs.top AND
			Not_AS.top AND
			Gotov_Vozb.top AND
			Reactornyi_P.top AND
			dP_kr1.top AND
			Auto_Rej.top AND
			CK_IM_Norm.top AND
			HAnd_Mode.top AND
			Impuls_Gaz.top THEN
			ppuFirst_for_I:=TRUE; ELSE ppuFirst_for_I:=FALSE; END_IF//ППУ имитация пуска


IF			BMP_Err.top AND
			Level_masla_Norm.top AND
			T_masla_Norm.top AND
			Net_AO_KC_SHKS04M.top AND
			EGPA_Stop.top AND
			Avt_SHU_vkl.top AND
			All_IM_Off.top AND
			Nalichie220_SHU_Ai.top AND
			BP_Norm.top AND
			Naprajenie_U_IM.top AND
			MV_Poloj_RolledON.top AND
			NOT MV_Poloj_RolledOFF.top AND
			NOTAnalogNS.top AND 
			Net_ASPS_Analogs.top AND
			Not_AS.top AND
			Gotov_Vozb.top AND
			Chastotnyi_P.top AND
			Auto_Rej.top AND
			CK_IM_Norm.top AND
			HAnd_Mode.top THEN
			ppuFirst_for_V_Ch:=TRUE; ELSE ppuFirst_for_V_Ch:=FALSE;  END_IF


IF			BMP_Err.top AND
			Level_masla_Norm.top AND
			T_masla_Norm.top AND
			Net_AO_KC_SHKS04M.top AND
			EGPA_Stop.top AND
			Avt_SHU_vkl.top AND
			All_IM_Off.top AND
			Nalichie220_SHU_Ai.top AND
			BP_Norm.top AND
			Naprajenie_U_IM.top AND
			MV_Poloj_RolledON.top AND
			NOT MV_Poloj_RolledOFF.top AND
			NOTAnalogNS.top AND 
			Net_ASPS_Analogs.top AND
			Not_AS.top AND
			Gotov_Vozb.top AND
			Reactornyi_P.top AND
			Auto_Rej.top AND
			CK_IM_Norm.top AND
			HAnd_Mode.top THEN
			ppuFirst_for_V_R:=TRUE; ELSE ppuFirst_for_V_R:=FALSE; END_IF
				

	IF		BMP_Err.top AND
			Level_masla_Norm.top AND
			T_masla_Norm.top AND
			Net_AO_KC_SHKS04M.top AND
			Avt_SHU_vkl.top AND
			Nalichie220_SHU_Ai.top AND
			BP_Norm.top AND
			Naprajenie_U_IM.top AND
			MV_Poloj_RolledON.top AND
			NOT MV_Poloj_RolledOFF.top AND
			NOTAnalogNS.top AND 
			Not_AS.top AND
			Gotov_Vozb.top AND
			Chastotnyi_P.top AND
			Auto_Rej.top AND
			HAnd_Mode.top AND ((algmanager.mode=modegpa.MODE_PUSKAP_Ch) OR (algmanager.mode=modegpa.MODE_PUSKPP_Ch) OR (algmanager.mode=modegpa.MODE_PUSKV_Ch)) THEN
			ppuSecond_V_Pusk_Ch:=	TRUE; ELSE ppuSecond_V_Pusk_Ch:= FALSE; END_IF


	IF		BMP_Err.top AND
			Level_masla_Norm.top AND
			T_masla_Norm.top AND
			Net_AO_KC_SHKS04M.top AND
			Avt_SHU_vkl.top AND
			Nalichie220_SHU_Ai.top AND
			BP_Norm.top AND
			Naprajenie_U_IM.top AND
			MV_Poloj_RolledON.top AND
			NOT MV_Poloj_RolledOFF.top AND
			NOTAnalogNS.top AND 
			Not_AS.top AND
			Gotov_Vozb.top AND
			Reactornyi_P.top AND
			Auto_Rej.top AND
			HAnd_Mode.top AND ((algmanager.mode=modegpa.MODE_PUSKAP_R) OR (algmanager.mode=modegpa.MODE_PUSKPP_R) OR (algmanager.mode=modegpa.MODE_PUSKV_R)) THEN
			ppuSecond_V_Pusk_R:=TRUE; ELSE ppuSecond_V_Pusk_R:=	FALSE; END_IF


	IF		BMP_Err.top AND
			Level_masla_Norm.top AND
			T_masla_Norm.top AND
			Net_AO_KC_SHKS04M.top AND
			Avt_SHU_vkl.top AND
			Nalichie220_SHU_Ai.top AND
			BP_Norm.top AND
			Naprajenie_U_IM.top AND
			MV_Poloj_RolledOFF.top AND
			NOT MV_Poloj_RolledON.top AND
			NOTAnalogNS.top AND 
			Not_AS.top AND
			Gotov_Vozb.top AND
			Reactornyi_P.top AND
			Auto_Rej.top AND
			HAnd_Mode.top AND (algmanager.mode=modegpa.MODE_I) THEN
			ppuSecond_I:=	TRUE; ELSE ppuSecond_I:= FALSE; END_IF	//ППУ для второго этапа пуска в режиме "имитация пуска"
			

